(* IEC 61131-3 sources: PortalRobot/Portal_robot/Device/application/FB (part 3) *)

(* ---- FB_ROBOT.st ---- *)
FUNCTION_BLOCK FB_ROBOT
VAR_INPUT

	stMachine_1_Command : ST_ROBOT_COMMAND; // Команда роботу от первого станка
	stMachine_2_Command : ST_ROBOT_COMMAND; // Команда роботу от второго станка
	stMachine_3_Command : ST_ROBOT_COMMAND; // Команда роботу от третьего станка
	stMagazineCommand   : ST_ROBOT_COMMAND; // Команда роботу от магазина
	stCellCommand       : ST_ROBOT_COMMAND; // Команда позиционирования от менеджера ячейки
	stHmiCommand        : ST_ROBOT_COMMAND; // Ручная команда роботу с HMI
	xReset              : BOOL; // Сброс ошибок робота
    xMode               : BOOL; // Режим робота: TRUE — Modbus, FALSE — SoftMotion
	xManual      		: BOOL; // 1 - ручной режим работы, 0 - автоматический режим работы
	xGlobalError        : BOOL; // Глобальная ошибка ячейки
	xModbusBusy         : BOOL; // Внешний робот выполняет команду
	xModbusDone         : BOOL; // Внешний робот завершил команду
	xModbusError        : BOOL; // Ошибка обмена или внешнего робота

    stPoint : ARRAY [0..GVL_POINT.iPointNumber] OF ST_POINT; // Глобальная таблица точек робота

    xSimBlankAvailable : BOOL; // Начальное наличие заготовки в модели захвата

END_VAR
VAR_OUTPUT
	Command       : ST_ROBOT_COMMAND; // Выбранная команда текущего цикла
	ModbusCommand : ST_ROBOT_COMMAND; // Команда внешнему роботу по Modbus
	Status        : ST_ROBOT_STATUS; // Рабочие статусы робота
	Diag          : ST_ROBOT_DIAG; // Состояние автомата и активная команда
	Error         : ST_ROBOT_ERRORS; // Активные и последние ошибки
	GripperDiag   : ST_GRIPPER_DIAG; // Диагностика внутреннего блока захвата
	GripperError  : ST_GRIPPER_ERRORS; // Активные и последние ошибки захвата
END_VAR
VAR
	fbMotionManager  : FB_MOTION_MANAGER; // Менеджер перемещения по точкам
    fbGripper        : FB_GRIPPER_SIMULATION; // Модель двухпозиционного захвата
	stGripperCommand : ST_GRIPPER_COMMAND; // Команда внутренней модели захвата

    eState        : E_ROBOT_STATE := E_ROBOT_STATE.IDLE; // Текущее состояние автомата робота
    eActiveAction : E_ROBOT_ACTION := E_ROBOT_ACTION.NONE; // Защёлкнутое действие
    eActivePoint  : E_POINT_NAME; // Защёлкнутая целевая точка

    xMotionExecute  : BOOL; // Запрос выполнения перемещения
    xGripperExecute : BOOL; // Запрос выполнения действия захвата
	xMagazineCommandActive : BOOL; // Активная команда получена от FB_MAGAZINE

END_VAR

VAR_IN_OUT
    stMotionManager : ST_MOTION_MANAGER; // Данные менеджера движения
    GroupData       : ST_AXIS_GROUP; // Данные группы осей XYZ
    stPointManager  : ST_POINT_MANAGER; // Данные проверки точки
END_VAR

VAR CONSTANT
	ERR_ROBOT_WRONG_ACTION : DWORD := DWORD#16#0000_0001; // Недопустимое действие робота
    ERR_ROBOT_MOTION       : DWORD := DWORD#16#0000_0002; // Ошибка менеджера движения
    ERR_ROBOT_GRIPPER      : DWORD := DWORD#16#0000_0004; // Ошибка захвата
    ERR_ROBOT_MODBUS_STUB  : DWORD := DWORD#16#0000_0008; // Ошибка внешнего робота или Modbus
    ERR_ROBOT_STOP         : DWORD := DWORD#16#0000_0010; // Остановка команды робота
	MASK_LOCAL_ERROR         : DWORD := ERR_ROBOT_WRONG_ACTION OR ERR_ROBOT_MODBUS_STUB; // Собственные первопричины робота
END_VAR

// --- BEGIN IMPLEMENTATION ---

// Команды по умолчанию
xMotionExecute := FALSE;
xGripperExecute := FALSE;
xMagazineCommandActive := FALSE;

Command.xExecute := FALSE;
Command.xStop := FALSE;
Command.xReset := FALSE;
Command.eAction := E_ROBOT_ACTION.NONE;
Command.eSetPoint := E_POINT_NAME.NONE;
Command.iTakeSlot := 0;
Command.iPutSlot := 0;

ModbusCommand.xExecute := FALSE;
ModbusCommand.xStop := FALSE;
ModbusCommand.xReset := xReset;
ModbusCommand.eAction := E_ROBOT_ACTION.NONE;
ModbusCommand.eSetPoint := E_POINT_NAME.NONE;
ModbusCommand.iTakeSlot := 0;
ModbusCommand.iPutSlot := 0;

//Определяем какой режим работы активен
IF NOT xManual THEN
	IF stCellCommand.xExecute OR stCellCommand.xStop THEN
		Command := stCellCommand;
	ELSIF stMachine_1_Command.xExecute THEN
		Command := stMachine_1_Command;
	ELSIF stMachine_2_Command.xExecute THEN
		Command := stMachine_2_Command;
	ELSIF stMachine_3_Command.xExecute THEN
		Command := stMachine_3_Command;
	ELSIF stMagazineCommand.xExecute OR stMagazineCommand.xStop THEN
		Command := stMagazineCommand;
		xMagazineCommandActive := TRUE;
	END_IF
ELSE
	IF stMagazineCommand.xExecute OR stMagazineCommand.xStop THEN
		Command := stMagazineCommand;
		xMagazineCommandActive := TRUE;
	ELSE
		Command := stHmiCommand;
	END_IF
END_IF;

Command.xReset := xReset;

// =====================================================
// Автомат FB_ROBOT
// =====================================================

CASE eState OF

    E_ROBOT_STATE.IDLE:

        Status.xBusy := FALSE;
        Status.xDone := FALSE;
        Status.xError := FALSE;

        IF Command.xExecute
		AND (xMagazineCommandActive
			OR ((Command.eSetPoint <> E_POINT_NAME.MAGAZINE_TAKE_DETAIL)
				AND (Command.eSetPoint <> E_POINT_NAME.MAGAZINE_PUT_DETAIL)
				AND (Command.eSetPoint <> E_POINT_NAME.MAGAZINE_CHANGE_DETAIL))) THEN
            eActiveAction := Command.eAction;
            eActivePoint := Command.eSetPoint;

            IF xMode THEN
                eState := E_ROBOT_STATE.MODBUS_STUB;

            ELSE
                CASE Command.eAction OF

                    E_ROBOT_ACTION.MOVE_TO_POINT:
                        eState := E_ROBOT_STATE.MOTION;

                    E_ROBOT_ACTION.UNCLAMP_1,
                    E_ROBOT_ACTION.CLAMP_1,
                    E_ROBOT_ACTION.UNCLAMP_2,
                    E_ROBOT_ACTION.CLAMP_2,
                    E_ROBOT_ACTION.ROTATE_TO_BLANK,
                    E_ROBOT_ACTION.ROTATE_TO_DETAIL:
                        eState := E_ROBOT_STATE.GRIPPER;

                ELSE
                    Error.dwErrorActive :=
                        Error.dwErrorActive OR ERR_ROBOT_WRONG_ACTION;

                    eState := E_ROBOT_STATE.ERROR;
                END_CASE;
            END_IF;
        END_IF;

    E_ROBOT_STATE.MOTION:

        Status.xBusy := TRUE;
        xMotionExecute := TRUE;

        IF Command.xStop OR xGlobalError THEN
            Error.dwErrorActive := Error.dwErrorActive OR ERR_ROBOT_STOP;
            eState := E_ROBOT_STATE.ERROR;

        ELSIF stMotionManager.Status.xError THEN
            Error.dwErrorActive := Error.dwErrorActive OR ERR_ROBOT_MOTION;
            eState := E_ROBOT_STATE.ERROR;

        ELSIF stMotionManager.Status.xDone THEN
            eState := E_ROBOT_STATE.DONE;
        END_IF;

    E_ROBOT_STATE.GRIPPER:

        Status.xBusy := TRUE;
        xGripperExecute := TRUE;

        IF Command.xStop OR xGlobalError THEN
            Error.dwErrorActive := Error.dwErrorActive OR ERR_ROBOT_STOP;
            eState := E_ROBOT_STATE.ERROR;

        ELSIF fbGripper.Status.xError THEN
            Error.dwErrorActive := Error.dwErrorActive OR ERR_ROBOT_GRIPPER;
            eState := E_ROBOT_STATE.ERROR;

        ELSIF fbGripper.Status.xDone THEN
            eState := E_ROBOT_STATE.DONE;
        END_IF;

    E_ROBOT_STATE.DONE:

        Status.xBusy := FALSE;
        Status.xDone := TRUE;

        CASE eActiveAction OF

            E_ROBOT_ACTION.MOVE_TO_POINT:
                xMotionExecute := TRUE;

            E_ROBOT_ACTION.UNCLAMP_1,
            E_ROBOT_ACTION.CLAMP_1,
            E_ROBOT_ACTION.UNCLAMP_2,
            E_ROBOT_ACTION.CLAMP_2,
            E_ROBOT_ACTION.ROTATE_TO_BLANK,
            E_ROBOT_ACTION.ROTATE_TO_DETAIL:
                xGripperExecute := TRUE;

        END_CASE;

        IF NOT Command.xExecute THEN
            Status.xDone := FALSE;
            eActiveAction := E_ROBOT_ACTION.NONE;
            eState := E_ROBOT_STATE.IDLE;
        END_IF;

    E_ROBOT_STATE.MODBUS_STUB:
		Status.xBusy := TRUE;
		ModbusCommand := Command;
		ModbusCommand.xExecute := TRUE;

		IF Command.xStop OR xGlobalError THEN
			ModbusCommand.xStop := TRUE;
			Error.dwErrorActive := Error.dwErrorActive OR ERR_ROBOT_STOP;
			eState := E_ROBOT_STATE.ERROR;
		ELSIF xModbusError THEN
			Error.dwErrorActive := Error.dwErrorActive OR ERR_ROBOT_MODBUS_STUB;
			eState := E_ROBOT_STATE.ERROR;
		ELSIF xModbusDone THEN
			eState := E_ROBOT_STATE.DONE;
		END_IF;

    E_ROBOT_STATE.ERROR:

        Status.xBusy := FALSE;
        Status.xDone := FALSE;
        Status.xError := TRUE;

        IF xReset
        AND NOT Command.xExecute
        AND NOT Command.xStop
        AND NOT xGlobalError
        AND NOT stMotionManager.Status.xError
		AND NOT fbGripper.Status.xError
		AND NOT xModbusError THEN

			Error.dwErrorLast := Error.dwErrorActive;
            Error.dwErrorActive := DWORD#0;
            Status.xError := FALSE;
            eActiveAction := E_ROBOT_ACTION.NONE;
            eState := E_ROBOT_STATE.IDLE;
        END_IF;

END_CASE;

// =====================================================
// Формирование команды FB_MOTION_MANAGER
// =====================================================

stMotionManager.Command.xExecute := xMotionExecute;
stMotionManager.Command.eTargetPoint := eActivePoint;
stMotionManager.Command.xReset := xReset;

// В ST_MOTION_MANAGER_COMMAND нет отдельного xStop.
// Поэтому Stop передаётся как ошибка верхнего уровня.
stMotionManager.Command.xGlobalError :=
    xGlobalError OR Command.xStop;

// =====================================================
// Вызов FB_MOTION_MANAGER
// =====================================================

fbMotionManager(
    stPoint := stPoint,
    xReset := xReset,
    stMotionManager := stMotionManager,
    GroupData := GroupData,
    stPointManager := stPointManager
);

// =====================================================
// Вызов FB_GRIPPER
// =====================================================

stGripperCommand.xExecute := xGripperExecute;
stGripperCommand.xReset := xReset;
stGripperCommand.eAction := eActiveAction;

fbGripper(
	Command := stGripperCommand,
	Diag => GripperDiag,
	Error => GripperError
);

// =====================================================
// Общие статусы
// =====================================================

Status.eCurrentPoint := stMotionManager.Status.eCurrentPoint;
Status.xGripper1Open :=
    fbGripper.Status.xGripper1Open;

Status.xGripper1Closed :=
    fbGripper.Status.xGripper1Closed;

Status.xGripper2Open :=
    fbGripper.Status.xGripper2Open;

Status.xGripper2Closed :=
    fbGripper.Status.xGripper2Closed;

Status.xRotatedToBlank :=
    fbGripper.Status.xRotatedToBlank;

Status.xRotatedToDetail :=
    fbGripper.Status.xRotatedToDetail;

Status.xBlankAvailable := Status.xGripper1Closed;
Status.xDetailAvailable := Status.xGripper2Closed;

Diag.eState := eState;
Diag.eActiveAction := eActiveAction;
Diag.eActivePoint := eActivePoint;
Error.dwAlarmActive := Error.dwErrorActive AND MASK_LOCAL_ERROR;
Status.xExternalError := (Error.dwErrorActive AND (ERR_ROBOT_MOTION OR ERR_ROBOT_GRIPPER)) <> DWORD#0;

IF Error.dwErrorActive <> DWORD#0 THEN
	Error.dwErrorLast := Error.dwErrorActive;
END_IF;

Error.stErrorActive := UpdateErrorView(dwError := Error.dwErrorActive);
Error.stErrorLast := UpdateErrorView(dwError := Error.dwErrorLast);

(* ---- FB_ROBOT_MODBUS.st ---- *)
{attribute 'no_assign'}
FUNCTION_BLOCK FB_ROBOT_MODBUS
VAR_INPUT
	xEnable          : BOOL; // Применён режим MODBUS_TCP
	xReconnect       : BOOL; // Настройки изменены, выполнить reconnect
	Config           : ST_ROBOT_MODBUS_CONFIG;
	Command          : ST_ROBOT_COMMAND; // Семантическая команда FB_ROBOT
END_VAR
VAR_OUTPUT
	Status           : ST_ROBOT_MODBUS_STATUS;
END_VAR
VAR_IN_OUT
	auiWriteRegisters : ARRAY [0..8] OF UINT; // Документные адреса 1001..1009
	auiReadRegisters  : ARRAY [0..16] OF UINT; // Документные адреса 1101..1117
END_VAR
VAR
	{attribute 'no_assign'}
	fbClient       : ModbusFB.ClientTCP;
	fbRead         : ModbusFB.ClientRequestReadHoldingRegisters;
	fbWrite        : ModbusFB.ClientRequestWriteMultipleRegisters;
	eState         : E_ROBOT_MODBUS_CLIENT_STATE := E_ROBOT_MODBUS_CLIENT_STATE.DISABLED;
	xConnect       : BOOL;
	xReadExecute   : BOOL;
	xWriteExecute  : BOOL;
	xStatusFresh   : BOOL;
	xCommandArmed  : BOOL;
	xCommandActive : BOOL;
	xWritePending  : BOOL;
	xHeartbeatChanged : BOOL;
	xHeartbeatSeen : BOOL;
	xPlcHeartbeatDue : BOOL;
	xStopPending   : BOOL;
	xResetPending  : BOOL;
	xControlClearPending : BOOL;
	rtStop         : R_TRIG;
	rtReset        : R_TRIG;
	rtReconnect    : R_TRIG;
	tonPoll        : TON;
	tonPlcHeartbeat: TON;
	tonRobotHeartbeat : TON;
	tonCommunicationGrace : TON;
	tonCommandTimeout : TON;
	tonReconnect   : TON;
	uiCommandSeq   : UINT;
	uiActiveSeq    : UINT;
	uiDecodedRobotHeartbeat : UINT; // Heartbeat из последнего завершённого FC03
	uiPositionXHigh : UINT; // Координаты из того же завершённого FC03-снимка
	uiPositionXLow  : UINT;
	uiPositionYHigh : UINT;
	uiPositionYLow  : UINT;
	uiPositionZHigh : UINT;
	uiPositionZLow  : UINT;
	uiPlcHeartbeat : UINT;
	uiLastRobotHeartbeat : UINT;
	uiCommandCode  : UINT;
	uiRegisterIndex : UINT;
	dwPositionRaw  : DWORD;
	diPositionRaw  : DINT;
	udiReplyTimeoutUs : UDINT;
END_VAR
VAR CONSTANT
	COMMAND_START_ITEM : UINT := UINT#1000; // Документный 1001
	STATUS_START_ITEM  : UINT := UINT#1100; // Документный 1101
	COMMAND_QUANTITY   : UINT := UINT#9;
	STATUS_QUANTITY    : UINT := UINT#17;
	PROTOCOL_VERSION   : UINT := UINT#3;
	STATUS_CONTROLLER_ON  : UINT := UINT#16#0001;
	STATUS_AUTOMATIC_MODE : UINT := UINT#16#0002;
	STATUS_REMOTE_ENABLED : UINT := UINT#16#0004;
	STATUS_DRIVES_ENABLED : UINT := UINT#16#0008;
	STATUS_HOMED          : UINT := UINT#16#0010;
	STATUS_EMERGENCY_STOP : UINT := UINT#16#0020;
	STATUS_ROBOT_ALARM    : UINT := UINT#16#0040;
	STATUS_ROBOT_READY    : UINT := UINT#16#0080;
	STATUS_POSITION_VALID : UINT := UINT#16#0100;
	STATUS_SIMULATOR_ACTIVE : UINT := UINT#16#0200;
END_VAR

// --- BEGIN IMPLEMENTATION ---

Status.xConfigValid := (Config.aIpAddress[0] > BYTE#0)
	AND (Config.aIpAddress[0] < BYTE#224)
	AND (Config.uiPort > UINT#0)
	AND (Config.uiUnitId <= UINT#255)
	AND (Config.tResponseTimeout >= T#50MS)
	AND (Config.tPollInterval >= T#10MS)
	AND (Config.tHeartbeatTimeout >= T#500MS)
	AND (Config.tCommandTimeout >= T#1S);

	udiReplyTimeoutUs := TIME_TO_UDINT(Config.tResponseTimeout) * UDINT#1000;
	rtStop(CLK := Command.xStop);
	rtReset(CLK := Command.xReset);
	rtReconnect(CLK := xReconnect);
	IF rtStop.Q THEN
		xStopPending := TRUE;
	END_IF;
	IF rtReset.Q THEN
		xResetPending := TRUE;
	END_IF;
xReadExecute := FALSE;
xWriteExecute := FALSE;
xHeartbeatChanged := FALSE;

fbClient(
	xConnect := xConnect,
	aIPaddr := Config.aIpAddress,
	uiPort := Config.uiPort,
	tConnnectTimeOut := Config.tHeartbeatTimeout
);

IF NOT xEnable OR NOT Status.xConfigValid THEN
	xConnect := FALSE;
	eState := E_ROBOT_MODBUS_CLIENT_STATE.DISABLED;
	xStatusFresh := FALSE;
	xCommandArmed := FALSE;
	xCommandActive := FALSE;
	xWritePending := FALSE;
	xStopPending := FALSE;
	xResetPending := FALSE;
	xControlClearPending := FALSE;
	xHeartbeatSeen := FALSE;
	xPlcHeartbeatDue := FALSE;
	uiActiveSeq := UINT#0;
	Status.xConnected := FALSE;
ELSE
	xConnect := TRUE;
	IF rtReconnect.Q THEN
		xConnect := FALSE;
		eState := E_ROBOT_MODBUS_CLIENT_STATE.RECONNECT_WAIT;
		xStatusFresh := FALSE;
		xCommandArmed := FALSE;
		xCommandActive := FALSE;
		xWritePending := FALSE;
		xControlClearPending := FALSE;
		xHeartbeatSeen := FALSE;
		xPlcHeartbeatDue := FALSE;
	END_IF;
END_IF;

CASE eState OF
	E_ROBOT_MODBUS_CLIENT_STATE.DISABLED:
		IF xEnable AND Status.xConfigValid THEN
			xConnect := TRUE;
			eState := E_ROBOT_MODBUS_CLIENT_STATE.CONNECTING;
		END_IF;

	E_ROBOT_MODBUS_CLIENT_STATE.CONNECTING:
		IF fbClient.xConnected THEN
			eState := E_ROBOT_MODBUS_CLIENT_STATE.INITIAL_READ;
		ELSIF fbClient.xError THEN
			Status.udiClientError := TO_UDINT(fbClient.eErrorID);
			xConnect := FALSE;
			eState := E_ROBOT_MODBUS_CLIENT_STATE.RECONNECT_WAIT;
		END_IF;

	E_ROBOT_MODBUS_CLIENT_STATE.INITIAL_READ:
		xReadExecute := TRUE;
		IF fbRead.xDone THEN
			xStatusFresh := TRUE;
			uiCommandSeq := auiReadRegisters[0];
			uiActiveSeq := UINT#0;
			uiPlcHeartbeat := UINT#0;
			uiLastRobotHeartbeat := auiReadRegisters[6];
			xHeartbeatSeen := FALSE;
			FOR uiRegisterIndex := UINT#0 TO UINT#8 DO
				auiWriteRegisters[uiRegisterIndex] := UINT#0;
			END_FOR;
			auiWriteRegisters[7] := uiCommandSeq;
			eState := E_ROBOT_MODBUS_CLIENT_STATE.INITIAL_READ_RELEASE;
		ELSIF fbRead.xError THEN
			Status.udiReadError := TO_UDINT(fbRead.eErrorID);
			xConnect := FALSE;
			eState := E_ROBOT_MODBUS_CLIENT_STATE.RECONNECT_WAIT;
		END_IF;

	E_ROBOT_MODBUS_CLIENT_STATE.INITIAL_READ_RELEASE:
		IF NOT fbRead.xBusy THEN
			eState := E_ROBOT_MODBUS_CLIENT_STATE.CLEAR_COMMAND;
		END_IF;

	E_ROBOT_MODBUS_CLIENT_STATE.CLEAR_COMMAND:
		xWriteExecute := TRUE;
		IF fbWrite.xDone THEN
			eState := E_ROBOT_MODBUS_CLIENT_STATE.CLEAR_COMMAND_RELEASE;
		ELSIF fbWrite.xError THEN
			Status.udiWriteError := TO_UDINT(fbWrite.eErrorID);
			xConnect := FALSE;
			eState := E_ROBOT_MODBUS_CLIENT_STATE.RECONNECT_WAIT;
		END_IF;

	E_ROBOT_MODBUS_CLIENT_STATE.CLEAR_COMMAND_RELEASE:
		IF NOT fbWrite.xBusy THEN
			xCommandArmed := NOT Command.xExecute;
			xCommandActive := FALSE;
			eState := E_ROBOT_MODBUS_CLIENT_STATE.READY;
		END_IF;

	E_ROBOT_MODBUS_CLIENT_STATE.READY:
		IF NOT fbClient.xConnected OR fbClient.xError THEN
			Status.udiClientError := TO_UDINT(fbClient.eErrorID);
			xConnect := FALSE;
			eState := E_ROBOT_MODBUS_CLIENT_STATE.RECONNECT_WAIT;
		ELSIF xStopPending THEN
			// Stop always preempts Reset and normal commands.
			// Execute снимается сразу: после принятого CommandSeq это не отменяет
			// команду, зато позволяет роботу выйти из DONE/ERROR/STOPPED в IDLE.
			// Без этого уже завершённая дискретная команда навечно удерживала
			// Execute=1, а xControlClearPending ждал недостижимый IDLE.
			auiWriteRegisters[0] := UINT#0;
			auiWriteRegisters[1] := UINT#0;
			auiWriteRegisters[2] := UINT#1;
			auiWriteRegisters[3] := UINT#0;
			auiWriteRegisters[4] := UINT#0;
			auiWriteRegisters[5] := UINT#0;
			auiWriteRegisters[6] := UINT#0;
			xStopPending := FALSE;
			xResetPending := FALSE;
			xControlClearPending := TRUE;
			xWritePending := TRUE;
		ELSIF xResetPending THEN
			// Reset обязан прервать незавершённую очистку Stop. Иначе
			// xControlClearPending имеет приоритет и защёлкнутый Reset никогда
			// не попадает в регистр 1004.
			auiWriteRegisters[0] := UINT#0;
			auiWriteRegisters[1] := UINT#0;
			auiWriteRegisters[2] := UINT#0;
			auiWriteRegisters[3] := UINT#1;
			auiWriteRegisters[4] := UINT#0;
			auiWriteRegisters[5] := UINT#0;
			auiWriteRegisters[6] := UINT#0;
			xCommandActive := FALSE;
			uiActiveSeq := UINT#0;
			xCommandArmed := FALSE;
			xResetPending := FALSE;
			xControlClearPending := TRUE;
			xWritePending := TRUE;
		ELSIF xControlClearPending THEN
			// Stop удерживается до STOPPED/IDLE, Reset — до снятия аварии. Так
			// импульс не потеряется между более медленными циклами программы робота.
			IF ((auiWriteRegisters[2] = UINT#1)
				AND ((Status.uiExecutionState = TO_UINT(E_ROBOT_MODBUS_EXECUTION_STATE.STOPPED))
					OR (Status.uiExecutionState = TO_UINT(E_ROBOT_MODBUS_EXECUTION_STATE.IDLE))))
			OR ((auiWriteRegisters[3] = UINT#1)
				AND NOT Status.xRobotAlarm
				AND (Status.uiExecutionState =
					TO_UINT(E_ROBOT_MODBUS_EXECUTION_STATE.IDLE))) THEN
				auiWriteRegisters[2] := UINT#0;
				auiWriteRegisters[3] := UINT#0;
				xCommandActive := FALSE;
				uiActiveSeq := UINT#0;
				// Верхний FB удерживает Execute до появления Busy. Поэтому после
				// подтверждённой очистки принимаем уже удерживаемую новую команду,
				// а не требуем ещё одного фронта от HMI.
				xCommandArmed := TRUE;
				xControlClearPending := FALSE;
				xWritePending := TRUE;
			END_IF;
		ELSIF Command.xExecute AND xCommandArmed AND NOT xCommandActive THEN
			uiCommandCode := UINT#0;
			CASE Command.eAction OF
				E_ROBOT_ACTION.MOVE_TO_POINT:
					CASE Command.eSetPoint OF
						E_POINT_NAME.MACHINE_1_ABOVE: uiCommandCode := UINT#10;
						E_POINT_NAME.MACHINE_1_INSIDE: uiCommandCode := UINT#11;
						E_POINT_NAME.MACHINE_1_CHUCK_APROACH: uiCommandCode := UINT#12;
						E_POINT_NAME.MACHINE_1_CHUCK_POSITION: uiCommandCode := UINT#13;
						E_POINT_NAME.MACHINE_2_ABOVE: uiCommandCode := UINT#14;
						E_POINT_NAME.MACHINE_2_INSIDE: uiCommandCode := UINT#15;
						E_POINT_NAME.MACHINE_2_CHUCK_APROACH: uiCommandCode := UINT#16;
						E_POINT_NAME.MACHINE_2_CHUCK_POSITION: uiCommandCode := UINT#17;
						E_POINT_NAME.MACHINE_3_ABOVE: uiCommandCode := UINT#18;
						E_POINT_NAME.MACHINE_3_INSIDE: uiCommandCode := UINT#19;
						E_POINT_NAME.MACHINE_3_CHUCK_APROACH: uiCommandCode := UINT#20;
						E_POINT_NAME.MACHINE_3_CHUCK_POSITION: uiCommandCode := UINT#21;
						E_POINT_NAME.HOME_SAFETY: uiCommandCode := UINT#22;
						E_POINT_NAME.MAGAZINE_SAFE: uiCommandCode := UINT#23;
						E_POINT_NAME.MAGAZINE_CHANGE: uiCommandCode := UINT#24;
						E_POINT_NAME.MAGAZINE_IN_SLOT: uiCommandCode := UINT#25;
					END_CASE;
				E_ROBOT_ACTION.UNCLAMP_1: uiCommandCode := UINT#2;
				E_ROBOT_ACTION.CLAMP_1: uiCommandCode := UINT#3;
				E_ROBOT_ACTION.UNCLAMP_2: uiCommandCode := UINT#4;
				E_ROBOT_ACTION.CLAMP_2: uiCommandCode := UINT#5;
				E_ROBOT_ACTION.ROTATE_TO_BLANK: uiCommandCode := UINT#6;
				E_ROBOT_ACTION.ROTATE_TO_DETAIL: uiCommandCode := UINT#7;
			END_CASE;

			IF uiCommandCode > UINT#0 THEN
				uiCommandSeq := uiCommandSeq + UINT#1;
				IF uiCommandSeq = UINT#0 THEN
					uiCommandSeq := UINT#1;
				END_IF;
				uiActiveSeq := uiCommandSeq;
				auiWriteRegisters[0] := uiCommandCode;
				auiWriteRegisters[1] := UINT#1;
				auiWriteRegisters[2] := UINT#0;
				auiWriteRegisters[3] := UINT#0;
				auiWriteRegisters[4] := SINT_TO_UINT(Command.iActiveSlot);
				auiWriteRegisters[5] := Command.uiMagazineId;
				auiWriteRegisters[6] := UINT#0;
				auiWriteRegisters[7] := uiCommandSeq;
				xCommandActive := TRUE;
				xCommandArmed := FALSE;
				xWritePending := TRUE;
			END_IF;
		ELSIF NOT Command.xExecute AND xCommandActive THEN
			auiWriteRegisters[0] := UINT#0;
			auiWriteRegisters[1] := UINT#0;
			auiWriteRegisters[2] := UINT#0;
			auiWriteRegisters[3] := UINT#0;
			auiWriteRegisters[4] := UINT#0;
			auiWriteRegisters[5] := UINT#0;
			auiWriteRegisters[6] := UINT#0;
			xCommandActive := FALSE;
			// CommandSeq в регистре сохраняется как последний использованный номер,
			// но завершённая транзакция больше не имеет права публиковать Done.
			// Повтор после Reset всегда получит новый ненулевой sequence.
			uiActiveSeq := UINT#0;
			xCommandArmed := TRUE;
			xWritePending := TRUE;
		ELSIF NOT Command.xExecute THEN
			xCommandArmed := TRUE;
		END_IF;

		IF xPlcHeartbeatDue THEN
			uiPlcHeartbeat := uiPlcHeartbeat + UINT#1;
			auiWriteRegisters[8] := uiPlcHeartbeat;
			xPlcHeartbeatDue := FALSE;
			xWritePending := TRUE;
		END_IF;

		IF xWritePending THEN
			eState := E_ROBOT_MODBUS_CLIENT_STATE.WRITE_COMMAND;
		ELSIF tonPoll.Q THEN
			eState := E_ROBOT_MODBUS_CLIENT_STATE.READ_STATUS;
		END_IF;

	E_ROBOT_MODBUS_CLIENT_STATE.WRITE_COMMAND:
		xWriteExecute := TRUE;
		IF fbWrite.xDone THEN
			xWritePending := FALSE;
			eState := E_ROBOT_MODBUS_CLIENT_STATE.WRITE_COMMAND_RELEASE;
		ELSIF fbWrite.xError THEN
			Status.udiWriteError := TO_UDINT(fbWrite.eErrorID);
			xConnect := FALSE;
			eState := E_ROBOT_MODBUS_CLIENT_STATE.RECONNECT_WAIT;
		END_IF;

	E_ROBOT_MODBUS_CLIENT_STATE.WRITE_COMMAND_RELEASE:
		IF NOT fbWrite.xBusy THEN
			eState := E_ROBOT_MODBUS_CLIENT_STATE.READ_STATUS;
		END_IF;

	E_ROBOT_MODBUS_CLIENT_STATE.READ_STATUS:
		xReadExecute := TRUE;
		IF fbRead.xDone THEN
			xStatusFresh := TRUE;
			eState := E_ROBOT_MODBUS_CLIENT_STATE.READ_STATUS_RELEASE;
		ELSIF fbRead.xError THEN
			Status.udiReadError := TO_UDINT(fbRead.eErrorID);
			xConnect := FALSE;
			eState := E_ROBOT_MODBUS_CLIENT_STATE.RECONNECT_WAIT;
		END_IF;

	E_ROBOT_MODBUS_CLIENT_STATE.READ_STATUS_RELEASE:
		IF NOT fbRead.xBusy THEN
			eState := E_ROBOT_MODBUS_CLIENT_STATE.READY;
		END_IF;

	E_ROBOT_MODBUS_CLIENT_STATE.RECONNECT_WAIT:
		xConnect := FALSE;
		xStatusFresh := FALSE;
		IF tonReconnect.Q THEN
			xConnect := TRUE;
			eState := E_ROBOT_MODBUS_CLIENT_STATE.CONNECTING;
		END_IF;
END_CASE;

fbRead(
	xExecute := xReadExecute,
	udiTimeOut := udiReplyTimeoutUs,
	rClient := fbClient,
	uiUnitId := Config.uiUnitId,
	udiReplyTimeout := udiReplyTimeoutUs,
	uiMaxRetries := UINT#1,
	uiStartItem := STATUS_START_ITEM,
	uiQuantity := STATUS_QUANTITY,
	pData := ADR(auiReadRegisters)
);
fbWrite(
	xExecute := xWriteExecute,
	udiTimeOut := udiReplyTimeoutUs,
	rClient := fbClient,
	uiUnitId := Config.uiUnitId,
	udiReplyTimeout := udiReplyTimeoutUs,
	uiMaxRetries := UINT#1,
	uiStartItem := COMMAND_START_ITEM,
	uiQuantity := COMMAND_QUANTITY,
	pData := ADR(auiWriteRegisters)
);

// FC03 может завершиться внутри вызова fbRead. Декодирование выполняется после
// вызова, чтобы технологический Status и сырые диагностические регистры всегда
// относились к одному и тому же снимку опроса.
IF fbRead.xDone THEN
	Status.uiAckSeq := auiReadRegisters[0];
	Status.uiExecutionState := auiReadRegisters[1];
	Status.uiResultCode := auiReadRegisters[2];
	Status.uiActiveCommand := auiReadRegisters[3];
	Status.uiCurrentPoint := auiReadRegisters[4];
	Status.uiGripperStatus := auiReadRegisters[5];
	Status.uiRobotHeartbeat := auiReadRegisters[6];
	Status.uiStatusWord := auiReadRegisters[7];
	Status.uiAlarmCode := auiReadRegisters[8];
	Status.uiOperationPhase := auiReadRegisters[15];
	Status.uiProtocolVersion := auiReadRegisters[16];
	uiDecodedRobotHeartbeat := auiReadRegisters[6];
	uiPositionXHigh := auiReadRegisters[9];
	uiPositionXLow := auiReadRegisters[10];
	uiPositionYHigh := auiReadRegisters[11];
	uiPositionYLow := auiReadRegisters[12];
	uiPositionZHigh := auiReadRegisters[13];
	uiPositionZLow := auiReadRegisters[14];
END_IF;

tonPoll(IN := eState = E_ROBOT_MODBUS_CLIENT_STATE.READY, PT := Config.tPollInterval);
// Heartbeat timer is independent of request states. The due latch prevents a pulse
// from being lost while FC03/FC16 is busy.
tonPlcHeartbeat(
	IN := xEnable AND fbClient.xConnected AND NOT tonPlcHeartbeat.Q,
	PT := T#100MS
);
IF tonPlcHeartbeat.Q THEN
	xPlcHeartbeatDue := TRUE;
END_IF;
tonReconnect(IN := eState = E_ROBOT_MODBUS_CLIENT_STATE.RECONNECT_WAIT, PT := T#1S);

Status.xConnected := fbClient.xConnected AND xConnect;
Status.xStatusFresh := xStatusFresh;

IF uiDecodedRobotHeartbeat <> uiLastRobotHeartbeat THEN
	uiLastRobotHeartbeat := uiDecodedRobotHeartbeat;
	xHeartbeatChanged := TRUE;
	xHeartbeatSeen := TRUE;
END_IF;
tonRobotHeartbeat(
	IN := xEnable AND xStatusFresh AND NOT xHeartbeatChanged,
	PT := Config.tHeartbeatTimeout
);
Status.xCommunicationAlive := Status.xConnected
	AND xStatusFresh
	AND xHeartbeatSeen
	AND NOT tonRobotHeartbeat.Q
	AND (Status.uiProtocolVersion = PROTOCOL_VERSION);
tonCommunicationGrace(
	IN := xEnable AND Status.xConfigValid AND NOT Status.xCommunicationAlive,
	PT := Config.tHeartbeatTimeout
);

Status.xControllerOn := (Status.uiStatusWord AND STATUS_CONTROLLER_ON) <> UINT#0;
Status.xAutomaticMode := (Status.uiStatusWord AND STATUS_AUTOMATIC_MODE) <> UINT#0;
Status.xRemoteEnabled := (Status.uiStatusWord AND STATUS_REMOTE_ENABLED) <> UINT#0;
Status.xDrivesEnabled := (Status.uiStatusWord AND STATUS_DRIVES_ENABLED) <> UINT#0;
Status.xHomed := (Status.uiStatusWord AND STATUS_HOMED) <> UINT#0;
Status.xEmergencyStop := (Status.uiStatusWord AND STATUS_EMERGENCY_STOP) <> UINT#0;
Status.xRobotAlarm := ((Status.uiStatusWord AND STATUS_ROBOT_ALARM) <> UINT#0)
	OR (Status.uiAlarmCode <> UINT#0);
Status.xPositionValid := (Status.uiStatusWord AND STATUS_POSITION_VALID) <> UINT#0;
Status.xSimulatorActive := (Status.uiStatusWord AND STATUS_SIMULATOR_ACTIVE) <> UINT#0;
Status.xReady := Status.xCommunicationAlive
	AND Status.xControllerOn
	AND Status.xAutomaticMode
	AND Status.xRemoteEnabled
	AND Status.xDrivesEnabled
	AND Status.xHomed
	AND Status.xPositionValid
	AND NOT Status.xEmergencyStop
	AND NOT Status.xRobotAlarm
	AND ((Status.uiStatusWord AND STATUS_ROBOT_READY) <> UINT#0);

Status.xDone := (uiActiveSeq <> UINT#0)
	AND xCommandActive
	AND (Status.uiAckSeq = uiActiveSeq)
	AND (Status.uiExecutionState = TO_UINT(E_ROBOT_MODBUS_EXECUTION_STATE.DONE))
	AND (Status.uiResultCode = UINT#0);
// Busy означает активную PLC-транзакцию, включая ожидание AckSeq. Благодаря
// этому FB_ROBOT обязательно увидит запуск новой команды до её terminal state.
Status.xBusy := (uiActiveSeq <> UINT#0)
	AND xCommandActive
	AND NOT Status.xDone
	AND NOT ((Status.uiAckSeq = uiActiveSeq)
		AND ((Status.uiExecutionState = TO_UINT(E_ROBOT_MODBUS_EXECUTION_STATE.ERROR))
			OR (Status.uiExecutionState = TO_UINT(E_ROBOT_MODBUS_EXECUTION_STATE.STOPPED))
			OR ((Status.uiExecutionState = TO_UINT(E_ROBOT_MODBUS_EXECUTION_STATE.DONE))
				AND (Status.uiResultCode <> UINT#0))));
tonCommandTimeout(
	IN := xCommandActive AND NOT Status.xDone,
	PT := Config.tCommandTimeout
);
Status.xCommandTimeout := tonCommandTimeout.Q;
Status.xError := tonCommunicationGrace.Q
	OR Status.xRobotAlarm
	OR Status.xCommandTimeout
	OR ((uiActiveSeq <> UINT#0)
		AND (Status.uiAckSeq = uiActiveSeq)
		AND ((Status.uiExecutionState = TO_UINT(E_ROBOT_MODBUS_EXECUTION_STATE.ERROR))
			OR ((Status.uiExecutionState = TO_UINT(E_ROBOT_MODBUS_EXECUTION_STATE.DONE))
				AND (Status.uiResultCode <> UINT#0))));

dwPositionRaw := SHL(UINT_TO_DWORD(uiPositionXHigh), 16)
	OR UINT_TO_DWORD(uiPositionXLow);
diPositionRaw := DWORD_TO_DINT(dwPositionRaw);
Status.lrActualX := DINT_TO_LREAL(diPositionRaw) / LREAL#10.0;
dwPositionRaw := SHL(UINT_TO_DWORD(uiPositionYHigh), 16)
	OR UINT_TO_DWORD(uiPositionYLow);
diPositionRaw := DWORD_TO_DINT(dwPositionRaw);
Status.lrActualY := DINT_TO_LREAL(diPositionRaw) / LREAL#10.0;
dwPositionRaw := SHL(UINT_TO_DWORD(uiPositionZHigh), 16)
	OR UINT_TO_DWORD(uiPositionZLow);
diPositionRaw := DWORD_TO_DINT(dwPositionRaw);
Status.lrActualZ := DINT_TO_LREAL(diPositionRaw) / LREAL#10.0;

(* ---- FB_SIMULATION_DYNAMIC_LIMITS.st ---- *)
FUNCTION_BLOCK FB_SIMULATION_DYNAMIC_LIMITS
VAR_INPUT
	xSimulationMode : BOOL; // Активна тестовая среда SIMULATION
	xSoftMotionMode : BOOL; // Роботом управляют локальные оси SoftMotion
	xAccelerationEnabled : BOOL; // Для следующего теста выбран ускоренный профиль
	xPrepareTest : BOOL; // Фронт подготовки следующего сценария
	uiRequestedFactor : UINT; // Запрошенное масштабирование времени 1..100
	xCellRunning : BOOL;
	xRobotBusy : BOOL;
	xMotionBusy : BOOL;
	xDrivesPowered : BOOL;
	xDrivesOff : BOOL;
	eGroupState : E_AXIS_GROUP_STATE;
	tTransactionTimeout : TIME := T#60S; // Общий предел Stop -> Disable -> Change -> Enable
END_VAR
VAR_OUTPUT
	xCellStopRequest : BOOL; // Сначала остановить технологический цикл
	xMotionStopRequest : BOOL; // Затем остановить движение группы
	xGroupDisableRequest : BOOL; // Перед изменением лимитов получить GroupDisabled
	xDrivesEnableRequest : BOOL; // После изменения вернуть штатную готовность
	xBusy : BOOL;
	xPending : BOOL; // Ползунок изменён; значение ждёт границы следующего теста
	xReadyForTest : BOOL; // Новый тест можно запускать
	xAccelerationActive : BOOL;
	uiAppliedFactor : UINT := UINT#1;
	xDone : BOOL;
	xError : BOOL;
	udiErrorId : UDINT;
END_VAR
VAR_IN_OUT
	AxisX : AXIS_REF_SM3;
	AxisY : AXIS_REF_SM3;
	AxisZ : AXIS_REF_SM3;
END_VAR
VAR CONSTANT
	STATE_IDLE : UINT := UINT#0;
	STATE_WAIT_STANDSTILL : UINT := UINT#10;
	STATE_WAIT_GROUP_DISABLED : UINT := UINT#20;
	STATE_CHANGE_X : UINT := UINT#30;
	STATE_CHANGE_Y : UINT := UINT#40;
	STATE_CHANGE_Z : UINT := UINT#50;
	STATE_PREPARE_ROLLBACK : UINT := UINT#55;
	STATE_WAIT_REENABLE : UINT := UINT#60;
	STATE_LOCKED_ERROR : UINT := UINT#90;
	ERR_INVALID_ORIGINAL_LIMITS : UDINT := UDINT#16#80010001;
	ERR_TRANSACTION_TIMEOUT : UDINT := UDINT#16#80010002;
	ERR_INVALID_STATE : UDINT := UDINT#16#80010003;
END_VAR
VAR
	rtPrepareTest : R_TRIG;
	tonTransaction : TON;
	uiState : UINT := UINT#0;
	uiAxis : UINT;
	uiDesiredFactor : UINT := UINT#1;
	uiTargetFactor : UINT := UINT#1;
	xOriginalLimitsSaved : BOOL;
	xOriginalLimitsValid : BOOL;
	xRestoreOnExit : BOOL;
	xRollback : BOOL;
	xReenableAfterChange : BOOL;

	alrOriginalVelocity : ARRAY [1..3] OF LREAL;
	alrOriginalAcceleration : ARRAY [1..3] OF LREAL;
	alrOriginalDeceleration : ARRAY [1..3] OF LREAL;
	alrOriginalJerk : ARRAY [1..3] OF LREAL;
	alrTargetVelocity : ARRAY [1..3] OF LREAL;
	alrTargetAcceleration : ARRAY [1..3] OF LREAL;
	alrTargetDeceleration : ARRAY [1..3] OF LREAL;
	alrTargetJerk : ARRAY [1..3] OF LREAL;
	lrFactor : LREAL;
	lrFactorSquared : LREAL;
	lrFactorCubed : LREAL;

	fbChangeX : SMC_ChangeDynamicLimits;
	fbChangeY : SMC_ChangeDynamicLimits;
	fbChangeZ : SMC_ChangeDynamicLimits;
END_VAR

// --- BEGIN IMPLEMENTATION ---

// Запрошенное значение разрешено менять когда угодно. Оно только создаёт
// pending-запрос; уже выполняемая траектория никогда не перепланируется.
uiDesiredFactor := MAX(UINT#1, MIN(UINT#100, uiRequestedFactor));
IF NOT (xSimulationMode AND xSoftMotionMode AND xAccelerationEnabled) THEN
	uiDesiredFactor := UINT#1;
END_IF;
rtPrepareTest(CLK := xPrepareTest);

xCellStopRequest := FALSE;
xMotionStopRequest := FALSE;
xGroupDisableRequest := FALSE;
xDrivesEnableRequest := FALSE;
xDone := FALSE;

// Штатные лимиты снимаются ровно при входе в SoftMotion-симуляцию, до первого
// масштабирования. Прямое редактирование AXIS_REF здесь не выполняется.
IF xSimulationMode AND xSoftMotionMode AND NOT xOriginalLimitsSaved THEN
	// Dynamic limits из конфигуратора оси находятся в fSWMax*. fMax* — это
	// remote limits самого привода и у виртуальной оси законно остаются нулями.
	alrOriginalVelocity[1] := AxisX.fSWMaxVelocity;
	alrOriginalAcceleration[1] := AxisX.fSWMaxAcceleration;
	alrOriginalDeceleration[1] := AxisX.fSWMaxDeceleration;
	alrOriginalJerk[1] := AxisX.fSWMaxJerk;
	alrOriginalVelocity[2] := AxisY.fSWMaxVelocity;
	alrOriginalAcceleration[2] := AxisY.fSWMaxAcceleration;
	alrOriginalDeceleration[2] := AxisY.fSWMaxDeceleration;
	alrOriginalJerk[2] := AxisY.fSWMaxJerk;
	alrOriginalVelocity[3] := AxisZ.fSWMaxVelocity;
	alrOriginalAcceleration[3] := AxisZ.fSWMaxAcceleration;
	alrOriginalDeceleration[3] := AxisZ.fSWMaxDeceleration;
	alrOriginalJerk[3] := AxisZ.fSWMaxJerk;

	IF alrOriginalVelocity[1] <= LREAL#0.0 THEN alrOriginalVelocity[1] := AxisX.fMaxVelocity; END_IF;
	IF alrOriginalAcceleration[1] <= LREAL#0.0 THEN alrOriginalAcceleration[1] := AxisX.fMaxAcceleration; END_IF;
	IF alrOriginalDeceleration[1] <= LREAL#0.0 THEN alrOriginalDeceleration[1] := AxisX.fMaxDeceleration; END_IF;
	IF alrOriginalJerk[1] <= LREAL#0.0 THEN alrOriginalJerk[1] := AxisX.fMaxJerk; END_IF;
	IF alrOriginalVelocity[2] <= LREAL#0.0 THEN alrOriginalVelocity[2] := AxisY.fMaxVelocity; END_IF;
	IF alrOriginalAcceleration[2] <= LREAL#0.0 THEN alrOriginalAcceleration[2] := AxisY.fMaxAcceleration; END_IF;
	IF alrOriginalDeceleration[2] <= LREAL#0.0 THEN alrOriginalDeceleration[2] := AxisY.fMaxDeceleration; END_IF;
	IF alrOriginalJerk[2] <= LREAL#0.0 THEN alrOriginalJerk[2] := AxisY.fMaxJerk; END_IF;
	IF alrOriginalVelocity[3] <= LREAL#0.0 THEN alrOriginalVelocity[3] := AxisZ.fMaxVelocity; END_IF;
	IF alrOriginalAcceleration[3] <= LREAL#0.0 THEN alrOriginalAcceleration[3] := AxisZ.fMaxAcceleration; END_IF;
	IF alrOriginalDeceleration[3] <= LREAL#0.0 THEN alrOriginalDeceleration[3] := AxisZ.fMaxDeceleration; END_IF;
	IF alrOriginalJerk[3] <= LREAL#0.0 THEN alrOriginalJerk[3] := AxisZ.fMaxJerk; END_IF;

	xOriginalLimitsValid := TRUE;
	FOR uiAxis := UINT#1 TO UINT#3 DO
		xOriginalLimitsValid := xOriginalLimitsValid
			AND (alrOriginalVelocity[uiAxis] > LREAL#0.0)
			AND (alrOriginalAcceleration[uiAxis] > LREAL#0.0)
			AND (alrOriginalDeceleration[uiAxis] > LREAL#0.0)
			AND (alrOriginalJerk[uiAxis] > LREAL#0.0);
	END_FOR;
	IF xOriginalLimitsValid THEN
		xOriginalLimitsSaved := TRUE;
		uiAppliedFactor := UINT#1;
		xError := FALSE;
		udiErrorId := UDINT#0;
	ELSIF rtPrepareTest.Q THEN
		// До подготовки теста просто ждём инициализацию осей; не защёлкиваем
		// ложную ошибку на первом цикле после переключения среды.
		xError := TRUE;
		udiErrorId := ERR_INVALID_ORIGINAL_LIMITS;
	END_IF;
END_IF;

// Ошибка чтения исходных лимитов не должна блокировать обычную ячейку после
// выхода из тестовой среды и не должна переживать Online Change этого исправления.
IF NOT xSimulationMode
AND NOT xOriginalLimitsSaved
AND (uiState = STATE_IDLE)
AND (udiErrorId = ERR_INVALID_ORIGINAL_LIMITS) THEN
	xError := FALSE;
	udiErrorId := UDINT#0;
END_IF;

xRestoreOnExit := xOriginalLimitsSaved
	AND (NOT xSimulationMode OR NOT xSoftMotionMode)
	AND (uiAppliedFactor <> UINT#1);
xPending := xOriginalLimitsSaved AND (uiDesiredFactor <> uiAppliedFactor);

// Один общий таймаут защищает всю транзакцию Stop -> Disable -> Change -> Enable.
tonTransaction(IN := uiState <> STATE_IDLE, PT := tTransactionTimeout);
IF tonTransaction.Q
AND (uiState <> STATE_IDLE)
AND (uiState <> STATE_LOCKED_ERROR) THEN
	xError := TRUE;
	udiErrorId := ERR_TRANSACTION_TIMEOUT;
	uiState := STATE_LOCKED_ERROR;
END_IF;

CASE uiState OF
	STATE_IDLE:
		xBusy := FALSE;
		// Возврат штатных лимитов при выходе из SIMULATION выполняется сразу.
		// Обычная ячейка не получит Start, пока транзакция не закончена.
		IF xRestoreOnExit THEN
			xError := FALSE;
			udiErrorId := UDINT#0;
			uiTargetFactor := UINT#1;
			xRollback := FALSE;
			xReenableAfterChange := xSoftMotionMode AND NOT xDrivesOff;
			xBusy := TRUE;
			uiState := STATE_WAIT_STANDSTILL;
		ELSIF rtPrepareTest.Q
		AND xSimulationMode
		AND xSoftMotionMode
		AND xPending
		AND NOT xCellRunning THEN
			xError := FALSE;
			udiErrorId := UDINT#0;
			uiTargetFactor := uiDesiredFactor;
			xRollback := FALSE;
			xReenableAfterChange := NOT xDrivesOff;
			xBusy := TRUE;
			uiState := STATE_WAIT_STANDSTILL;
		ELSIF NOT xSimulationMode
		AND xOriginalLimitsSaved
		AND (uiAppliedFactor = UINT#1) THEN
			// Лимиты не менялись либо уже успешно восстановлены.
			xOriginalLimitsSaved := FALSE;
		END_IF;

	STATE_WAIT_STANDSTILL:
		xBusy := TRUE;
		xCellStopRequest := xCellRunning;
		xMotionStopRequest := xMotionBusy OR xRobotBusy;
		IF NOT xCellRunning AND NOT xMotionBusy AND NOT xRobotBusy THEN
			uiState := STATE_WAIT_GROUP_DISABLED;
		END_IF;

	STATE_WAIT_GROUP_DISABLED:
		xBusy := TRUE;
		xGroupDisableRequest := NOT xDrivesOff;
		IF xDrivesOff AND (eGroupState = E_AXIS_GROUP_STATE.DISABLED) THEN
			IF xRollback THEN
				FOR uiAxis := UINT#1 TO UINT#3 DO
					alrTargetVelocity[uiAxis] := alrOriginalVelocity[uiAxis];
					alrTargetAcceleration[uiAxis] := alrOriginalAcceleration[uiAxis];
					alrTargetDeceleration[uiAxis] := alrOriginalDeceleration[uiAxis];
					alrTargetJerk[uiAxis] := alrOriginalJerk[uiAxis];
				END_FOR;
			ELSE
				lrFactor := UINT_TO_LREAL(uiTargetFactor);
				lrFactorSquared := lrFactor * lrFactor;
				lrFactorCubed := lrFactorSquared * lrFactor;
				alrTargetVelocity[1] := alrOriginalVelocity[1] * lrFactor;
				alrTargetAcceleration[1] := alrOriginalAcceleration[1] * lrFactorSquared;
				alrTargetDeceleration[1] := alrOriginalDeceleration[1] * lrFactorSquared;
				alrTargetJerk[1] := alrOriginalJerk[1] * lrFactorCubed;
				alrTargetVelocity[2] := alrOriginalVelocity[2] * lrFactor;
				alrTargetAcceleration[2] := alrOriginalAcceleration[2] * lrFactorSquared;
				alrTargetDeceleration[2] := alrOriginalDeceleration[2] * lrFactorSquared;
				alrTargetJerk[2] := alrOriginalJerk[2] * lrFactorCubed;
				alrTargetVelocity[3] := alrOriginalVelocity[3] * lrFactor;
				alrTargetAcceleration[3] := alrOriginalAcceleration[3] * lrFactorSquared;
				alrTargetDeceleration[3] := alrOriginalDeceleration[3] * lrFactorSquared;
				alrTargetJerk[3] := alrOriginalJerk[3] * lrFactorCubed;
			END_IF;
			uiState := STATE_CHANGE_X;
		END_IF;

	STATE_CHANGE_X:
		xBusy := TRUE;
		IF fbChangeX.bError THEN
			xError := TRUE;
			udiErrorId := TO_UDINT(fbChangeX.ErrorID);
			IF xRollback THEN uiState := STATE_LOCKED_ERROR;
			ELSE uiState := STATE_PREPARE_ROLLBACK; END_IF;
		ELSIF fbChangeX.bDone THEN
			uiState := STATE_CHANGE_Y;
		END_IF;

	STATE_CHANGE_Y:
		xBusy := TRUE;
		IF fbChangeY.bError THEN
			xError := TRUE;
			udiErrorId := TO_UDINT(fbChangeY.ErrorID);
			IF xRollback THEN uiState := STATE_LOCKED_ERROR;
			ELSE uiState := STATE_PREPARE_ROLLBACK; END_IF;
		ELSIF fbChangeY.bDone THEN
			uiState := STATE_CHANGE_Z;
		END_IF;

	STATE_CHANGE_Z:
		xBusy := TRUE;
		IF fbChangeZ.bError THEN
			xError := TRUE;
			udiErrorId := TO_UDINT(fbChangeZ.ErrorID);
			IF xRollback THEN uiState := STATE_LOCKED_ERROR;
			ELSE uiState := STATE_PREPARE_ROLLBACK; END_IF;
		ELSIF fbChangeZ.bDone THEN
			IF xReenableAfterChange THEN
				uiState := STATE_WAIT_REENABLE;
			ELSE
				IF xRollback THEN uiAppliedFactor := UINT#1;
				ELSE uiAppliedFactor := uiTargetFactor; END_IF;
				xDone := NOT xRollback;
				xBusy := FALSE;
				uiState := STATE_IDLE;
			END_IF;
		END_IF;

	STATE_PREPARE_ROLLBACK:
		// Один цикл с Execute=FALSE создаёт корректный новый фронт для X.
		xBusy := TRUE;
		xRollback := TRUE;
		uiState := STATE_WAIT_GROUP_DISABLED;

	STATE_WAIT_REENABLE:
		xBusy := TRUE;
		xDrivesEnableRequest := TRUE;
		IF xDrivesPowered AND (eGroupState = E_AXIS_GROUP_STATE.READY) THEN
			IF xRollback THEN uiAppliedFactor := UINT#1;
			ELSE uiAppliedFactor := uiTargetFactor; END_IF;
			xDone := NOT xRollback;
			xBusy := FALSE;
			uiState := STATE_IDLE;
		END_IF;

	STATE_LOCKED_ERROR:
		// При неизвестном/неустранимом результате оставляем группу отключённой.
		// Следующий Start заблокирован, пока инженер не устранит причину.
		xBusy := FALSE;
		xGroupDisableRequest := NOT xDrivesOff;

ELSE
	xError := TRUE;
	udiErrorId := ERR_INVALID_STATE;
	uiState := STATE_LOCKED_ERROR;
END_CASE;

fbChangeX(
	Axis := AxisX,
	bExecute := uiState = STATE_CHANGE_X,
	fMaxVelocity := alrTargetVelocity[1],
	fMaxAcceleration := alrTargetAcceleration[1],
	fMaxDeceleration := alrTargetDeceleration[1],
	fMaxJerk := alrTargetJerk[1]
);
fbChangeY(
	Axis := AxisY,
	bExecute := uiState = STATE_CHANGE_Y,
	fMaxVelocity := alrTargetVelocity[2],
	fMaxAcceleration := alrTargetAcceleration[2],
	fMaxDeceleration := alrTargetDeceleration[2],
	fMaxJerk := alrTargetJerk[2]
);
fbChangeZ(
	Axis := AxisZ,
	bExecute := uiState = STATE_CHANGE_Z,
	fMaxVelocity := alrTargetVelocity[3],
	fMaxAcceleration := alrTargetAcceleration[3],
	fMaxDeceleration := alrTargetDeceleration[3],
	fMaxJerk := alrTargetJerk[3]
);

xPending := xOriginalLimitsSaved AND (uiDesiredFactor <> uiAppliedFactor);
xAccelerationActive := xSimulationMode AND xSoftMotionMode
	AND (uiAppliedFactor > UINT#1) AND NOT xError;
xReadyForTest := NOT xBusy AND NOT xError
	AND (NOT (xSimulationMode AND xSoftMotionMode AND xAccelerationEnabled) OR NOT xPending);

(* ---- FB_TWO_PALLET.st ---- *)
FUNCTION_BLOCK FB_TWO_PALLET
VAR_INPUT
	xSelected : BOOL;
	xManual : BOOL;
	xSafe : BOOL;
	xRobotClear : BOOL; // Окно планировщика и освобождение зоны для обмена в автоматическом режиме
	xRobotIdle : BOOL; // Останов робота без проверки точек, интерфейса и зоны магазина
	xRobotOperation : BOOL; // Текущая или уже выданная операция с этим магазином
	xRobotGeometryReady : BOOL; // Точки робота нужны для работы ячейки, но не для включения магазина
	xRobotMagazineReady : BOOL; // Ошибки и геометрия магазина; содержимое не блокирует включение
	xConnection : BOOL;
	xStopRequest : BOOL;
	xAutoSwap : BOOL;
	xOtherLoaded : BOOL;
	xActivePalletEditAllowed : BOOL;
	xConfigurationChanged : BOOL;
	xExternalCommandRejected : BOOL;
	Command : ST_TWO_PALLET_COMMAND;
	Config : ST_TWO_PALLET_CONFIG;
	Input : ST_TWO_PALLET_INPUT;
END_VAR
VAR_OUTPUT
	Status : ST_TWO_PALLET_STATUS;
	Diag : ST_TWO_PALLET_DIAG;
	Error : ST_TWO_PALLET_ERRORS;
	Output : ST_TWO_PALLET_OUTPUT;
END_VAR
VAR
	ePreviousState : E_TWO_PALLET_STATE := E_TWO_PALLET_STATE.IDLE;
	uiFrom : UINT;
	uiTo : UINT;
	uiSelected : UINT;
	uiCandidate : UINT;
	uiPreviousCandidate : UINT;
	uiConfirmedCandidate : UINT;
	uiManualSelected : UINT;
	uiJogDirection : UINT;
	uiSignals : UINT;
	uiSelectedSignals : UINT;
	uiTargetSignals : UINT;
	xPreviousBaseValid : BOOL;
	xConfigValid : BOOL;
	xContradiction : BOOL;
	xPairValid : BOOL;
	xWork : BOOL;
	xExchange : BOOL;
	xIdle : BOOL;
	xBase : BOOL;
	xRecovery : BOOL;
	xPneumaticBase : BOOL;
	xPneumaticRecovery : BOOL;
	xManualPneumaticState : BOOL;
	xAutomaticState : BOOL;
	xAxisMotionState : BOOL;
	xManualState : BOOL;
	xAutoSwapAllowed : BOOL;
	xExchangeStartedManual : BOOL; // Обмен начат в ручном режиме: без проверки роботной зоны/точек
	xCommandPresent : BOOL;
	xAccepted : BOOL;
	xStateEntry : BOOL;
	xSeenMotion : BOOL;
	xSeenDone : BOOL;
	xLiftUpCommand : BOOL;
	xLiftDownCommand : BOOL;
	xSelectCommand : BOOL;
	xManualLockCommand : BOOL;
	xManualStopCommand : BOOL;
	xManualLockOutTarget : BOOL;
	xManualStopOutTarget : BOOL;
	xLockOutTarget : BOOL;
	xStopOutTarget : BOOL;
	xStartupInitialized : BOOL;
	xTrustedAtScanStart : BOOL;
	lrWork : LREAL;
	lrTarget : LREAL;
	lrSpan : LREAL;
	rTravel : REAL;
	tStateLimit : TIME;
	tonState : TON;
	tonCoil : TON;
	tonJogLease : TON;
	dwPreviousError : DWORD;
END_VAR
VAR CONSTANT
	ERR_DRIVE : DWORD := DWORD#16#100;
	ERR_SENSOR_CONTRADICTION : DWORD := DWORD#16#200;
	ERR_CYLINDER_TIMEOUT : DWORD := DWORD#16#400;
	ERR_MOTION_TIMEOUT : DWORD := DWORD#16#800;
	ERR_LOGIC : DWORD := DWORD#16#1000;
	ERR_SEQUENCE_INTERRUPTED : DWORD := DWORD#16#2000;
	WRN_COMMAND_REJECTED : UINT := UINT#30;
	WRN_START_REJECTED_BY_OPERATOR : UINT := UINT#31;
	JOG_POSITIVE : UINT := UINT#1;
	JOG_NEGATIVE : UINT := UINT#2;
END_VAR

// --- BEGIN IMPLEMENTATION ---

// Шаги, разрешения и подтверждение положения не восстанавливаются после старта PLC.
IF NOT xStartupInitialized THEN
	Diag.eState := E_TWO_PALLET_STATE.IDLE;
	ePreviousState := E_TWO_PALLET_STATE.IDLE;
	Status.xConfirmed := FALSE;
	Status.xEnabled := FALSE;
	xStartupInitialized := TRUE;
END_IF;

Status.xCompleted := FALSE;
Status.Input := Input;
xTrustedAtScanStart := Status.xConfirmed;

// Все выходные команды импульсные или формируются заново на каждом скане.
Output.xPowerOn := FALSE;
Output.xPowerOff := FALSE;
Output.xDriveReset := FALSE;
Output.xHome := FALSE;
Output.xMove := FALSE;
Output.xStop := FALSE;
Output.xJogPositive := FALSE;
Output.xJogNegative := FALSE;
Output.xTeachOperator := FALSE;
Output.xTeachWork := FALSE;
xLiftUpCommand := FALSE;
xLiftDownCommand := FALSE;
xSelectCommand := FALSE;
xManualLockCommand := FALSE;
xManualStopCommand := FALSE;

// Конфигурация механизма.
xConfigValid := Config.xConfigured
	AND Config.xSignalPatternsConfigured
	AND IsSignalConfigurationValid(uiP1Signals := Config.uiP1Signals, uiP2Signals := Config.uiP2Signals)
	AND (Config.lrTolerance > 0.0)
	AND (Config.lrTolerance <= 20.0)
	AND (ABS(Config.lrWorkP1 - Config.lrExchange) > 2.0 * Config.lrTolerance)
	AND (ABS(Config.lrWorkP2 - Config.lrExchange) > 2.0 * Config.lrTolerance)
	AND ((Config.lrWorkP1 - Config.lrExchange) * (Config.lrWorkP2 - Config.lrExchange) > 0.0)
	AND (Config.lrVelocity > 0.0)
	AND (Config.lrAcceleration > 0.0)
	AND (Config.lrDeceleration > 0.0)
	AND (Config.lrJerk > 0.0)
	AND (Config.tPulse >= T#50MS)
	AND (Config.tCylinder > Config.tPulse)
	AND (Config.tMove > T#0S)
	AND (Config.tHome > T#0S);
Status.xConfigValid := xConfigValid;

// Фактическое состояние пневматики и каретки.
xContradiction := (Input.xLiftUp AND Input.xLiftDown)
	OR (Input.xLockIn AND Input.xLockOut)
	OR (Input.xStopIn AND Input.xStopOut)
	OR (Input.xLimitNegative AND Input.xLimitPositive);
xPairValid := (Input.xLockIn XOR Input.xLockOut)
	AND (Input.xStopIn XOR Input.xStopOut);

uiSignals := UINT#0;
IF Input.xLiftDown THEN uiSignals := uiSignals OR UINT#1; END_IF;
IF Input.xLiftUp THEN uiSignals := uiSignals OR UINT#2; END_IF;
IF Input.xLockIn THEN uiSignals := uiSignals OR UINT#4; END_IF;
IF Input.xLockOut THEN uiSignals := uiSignals OR UINT#8; END_IF;
IF Input.xStopIn THEN uiSignals := uiSignals OR UINT#16; END_IF;
IF Input.xStopOut THEN uiSignals := uiSignals OR UINT#32; END_IF;

uiSelected := UINT#0;
IF xPairValid THEN
	IF (uiSignals AND UINT#60) = (Config.uiP1Signals AND UINT#60) THEN
		uiSelected := UINT#1;
	ELSIF (uiSignals AND UINT#60) = (Config.uiP2Signals AND UINT#60) THEN
		uiSelected := UINT#2;
	END_IF;
END_IF;
xPairValid := xPairValid AND (uiSelected <> UINT#0);

lrWork := Config.lrWorkP1;
uiSelectedSignals := Config.uiP1Signals;
IF uiSelected = UINT#2 THEN
	lrWork := Config.lrWorkP2;
	uiSelectedSignals := Config.uiP2Signals;
END_IF;

xWork := xConfigValid
	AND Input.xHomed
	AND Input.xStandstill
	AND xPairValid
	AND (ABS(Input.lrPosition - lrWork) <= Config.lrTolerance);
xExchange := xConfigValid
	AND Input.xHomed
	AND Input.xStandstill
	AND (ABS(Input.lrPosition - Config.lrExchange) <= Config.lrTolerance);

uiCandidate := UINT#0;
IF xWork
	AND (uiSignals = uiSelectedSignals)
	AND NOT xContradiction
	AND NOT Input.xDriveError
	AND NOT Status.xHomeRequired THEN
	uiCandidate := uiSelected;
END_IF;

xIdle := Diag.eState = E_TWO_PALLET_STATE.IDLE;
xAutomaticState := (Diag.eState = E_TWO_PALLET_STATE.AUTO_LOWER)
	OR (Diag.eState = E_TWO_PALLET_STATE.AUTO_MOVE_TO_EXCHANGE)
	OR (Diag.eState = E_TWO_PALLET_STATE.AUTO_SELECT_PALLET)
	OR (Diag.eState = E_TWO_PALLET_STATE.AUTO_MOVE_TO_WORK)
	OR (Diag.eState = E_TWO_PALLET_STATE.AUTO_RAISE);
xAxisMotionState := (Diag.eState = E_TWO_PALLET_STATE.AUTO_MOVE_TO_EXCHANGE)
	OR (Diag.eState = E_TWO_PALLET_STATE.AUTO_MOVE_TO_WORK)
	OR (Diag.eState = E_TWO_PALLET_STATE.MANUAL_MOVE)
	OR (Diag.eState = E_TWO_PALLET_STATE.MANUAL_HOME)
	OR (Diag.eState = E_TWO_PALLET_STATE.MANUAL_JOG);
xManualState := (Diag.eState = E_TWO_PALLET_STATE.MANUAL_LOWER)
	OR (Diag.eState = E_TWO_PALLET_STATE.MANUAL_RAISE)
	OR (Diag.eState = E_TWO_PALLET_STATE.MANUAL_SELECT_PALLET)
	OR (Diag.eState = E_TWO_PALLET_STATE.MANUAL_MOVE)
	OR (Diag.eState = E_TWO_PALLET_STATE.MANUAL_HOME)
	OR (Diag.eState = E_TWO_PALLET_STATE.MANUAL_JOG)
	OR (Diag.eState = E_TWO_PALLET_STATE.MANUAL_LOCK)
	OR (Diag.eState = E_TWO_PALLET_STATE.MANUAL_STOP);
xManualPneumaticState := (Diag.eState = E_TWO_PALLET_STATE.MANUAL_LOWER)
	OR (Diag.eState = E_TWO_PALLET_STATE.MANUAL_LOCK)
	OR (Diag.eState = E_TWO_PALLET_STATE.MANUAL_STOP);

xBase := xSelected
	AND xConfigValid
	AND Input.xIoMapped
	AND Input.xAxisBound
	AND xSafe
	AND NOT xRobotOperation;
xRecovery := xBase
	AND xManual
	AND xConnection
	AND xIdle
	AND Input.xStandstill;
xPneumaticBase := xSelected
	AND xManual
	AND xSafe
	AND NOT xRobotOperation
	AND Input.xIoMapped
	AND Input.xStandstill;
xPneumaticRecovery := xPneumaticBase AND xIdle;

Status.uiCandidate := uiCandidate;
Status.uiSelected := uiSelected;

// Любое изменение достоверной расстановки аннулирует старое подтверждение.
IF (uiCandidate <> uiPreviousCandidate) OR (xBase <> xPreviousBaseValid) THEN
	Status.udiRevision := Status.udiRevision + UDINT#1;
	IF Status.udiRevision = UDINT#0 THEN
		Status.udiRevision := UDINT#1;
	END_IF;
END_IF;
uiPreviousCandidate := uiCandidate;
xPreviousBaseValid := xBase;

IF xConfigurationChanged THEN
	Status.xConfirmed := FALSE;
	Status.xEnabled := FALSE;
	Status.udiRevision := Status.udiRevision + UDINT#1;
	IF Status.udiRevision = UDINT#0 THEN
		Status.udiRevision := UDINT#1;
	END_IF;
END_IF;

IF NOT xSelected
	OR NOT xSafe
	OR NOT Input.xAxisBound
	OR NOT Input.xIoMapped
	OR NOT xConfigValid
	OR Input.xDriveError
	OR NOT Input.xPowered
	OR (xIdle AND (uiCandidate <> uiConfirmedCandidate)) THEN
	Status.xConfirmed := FALSE;
END_IF;
// Пропадание heartbeat выключает автоматическую обработку, но само по себе
// не перемещает механику и не стирает уже проверенную идентичность палет.
IF NOT xConnection THEN Status.xEnabled := FALSE; END_IF;

// Первая невыполненная предпосылка для HMI.
Diag.uiReason := UINT#0;
IF NOT xSelected THEN
	Diag.uiReason := UINT#1;
ELSIF NOT xConfigValid THEN
	Diag.uiReason := UINT#2;
ELSIF NOT Input.xAxisBound OR NOT Input.xIoMapped THEN
	Diag.uiReason := UINT#3;
ELSIF NOT xSafe THEN
	Diag.uiReason := UINT#4;
ELSIF NOT xConnection THEN
	Diag.uiReason := UINT#17;
ELSIF Input.xDriveError THEN
	Diag.uiReason := UINT#6;
ELSIF Error.dwErrorActive <> DWORD#0 THEN
	Diag.uiReason := UINT#19;
ELSIF NOT Input.xPowered THEN
	Diag.uiReason := UINT#18;
ELSIF xContradiction THEN
	Diag.uiReason := UINT#7;
ELSIF Status.xHomeRequired OR NOT Input.xHomed THEN
	Diag.uiReason := UINT#8;
ELSIF NOT xPairValid THEN
	Diag.uiReason := UINT#9;
ELSIF NOT Input.xStandstill THEN
	Diag.uiReason := UINT#10;
ELSIF NOT xWork THEN
	Diag.uiReason := UINT#11;
ELSIF uiSignals <> uiSelectedSignals THEN
	Diag.uiReason := UINT#12;
ELSIF NOT xIdle THEN
	Diag.uiReason := UINT#22;
ELSIF NOT xRobotMagazineReady THEN
	Diag.uiReason := UINT#16;
ELSIF NOT Status.xConfirmed AND NOT xManual THEN
	Diag.uiReason := UINT#20;
ELSIF NOT Status.xConfirmed THEN
	Diag.uiReason := UINT#13;
END_IF;

// Аварии механизма: биты 8..13 зарезервированы в MAGAZINE_LOGIC_1/2.
IF xSelected AND Input.xDriveError THEN
	Error.dwErrorActive := Error.dwErrorActive OR ERR_DRIVE;
	Status.xHomeRequired := TRUE;
END_IF;

IF xSelected AND xContradiction THEN
	Error.dwErrorActive := Error.dwErrorActive OR ERR_SENSOR_CONTRADICTION;
END_IF;

IF xSelected
	AND NOT xIdle
	AND (((NOT xBase) AND NOT (xManualPneumaticState AND xPneumaticBase))
		OR ((NOT xConnection) AND NOT xManualPneumaticState) OR xStopRequest
		OR (xAutomaticState AND ((xExchangeStartedManual AND (NOT xManual OR NOT xRobotIdle))
			OR (NOT xExchangeStartedManual AND NOT xRobotClear)))) THEN
	Error.dwErrorActive := Error.dwErrorActive OR ERR_SEQUENCE_INTERRUPTED;
	Diag.eState := E_TWO_PALLET_STATE.IDLE;
	Output.xStop := TRUE;
END_IF;

IF xSelected AND (xTrustedAtScanStart OR xAutomaticState) THEN
	IF ((Diag.eState <> E_TWO_PALLET_STATE.AUTO_SELECT_PALLET) AND NOT xPairValid)
		OR (((Diag.eState = E_TWO_PALLET_STATE.AUTO_MOVE_TO_EXCHANGE)
			OR (Diag.eState = E_TWO_PALLET_STATE.AUTO_MOVE_TO_WORK))
			AND (NOT Input.xLiftDown OR Input.xLiftUp))
		OR (xIdle AND (uiCandidate = UINT#0)) THEN
		Error.dwErrorActive := Error.dwErrorActive OR ERR_LOGIC;
	END_IF;
END_IF;

IF xSelected
	AND xTrustedAtScanStart
	AND (NOT xSafe
		OR NOT Input.xAxisBound
		OR NOT Input.xIoMapped
		OR NOT Input.xPowered) THEN
	Error.dwErrorActive := Error.dwErrorActive OR ERR_SEQUENCE_INTERRUPTED;
END_IF;

IF xSelected
	AND ((xContradiction AND NOT xIdle AND NOT xManualPneumaticState)
		OR (Input.xDriveError AND xAxisMotionState)) THEN
	Diag.eState := E_TWO_PALLET_STATE.IDLE;
	Output.xStop := TRUE;
END_IF;

IF xSelected AND NOT Input.xPowered AND (xAutomaticState OR xAxisMotionState) THEN
	Error.dwErrorActive := Error.dwErrorActive OR ERR_SEQUENCE_INTERRUPTED;
	Status.xHomeRequired := TRUE;
	Diag.eState := E_TWO_PALLET_STATE.IDLE;
	Output.xStop := TRUE;
END_IF;

IF Error.dwErrorActive <> DWORD#0 THEN
	Status.xEnabled := FALSE;
	Status.xConfirmed := FALSE;
	IF xAutomaticState THEN
		Diag.eState := E_TWO_PALLET_STATE.IDLE;
		Output.xStop := TRUE;
	END_IF;
END_IF;

// Разрешения считаются только владельцем механизма.
Status.xConfirmAllowed := xRecovery
	AND Input.xPowered
	AND (uiCandidate <> UINT#0)
	AND (Error.dwErrorActive = DWORD#0);
Status.xStartAllowed := Status.xConfirmAllowed
	AND xRobotMagazineReady;
Status.xEnableAllowed := xBase
	AND xConnection
	AND xIdle
	AND Status.xConfirmed
	AND xRobotMagazineReady
	AND (uiCandidate = Status.uiRobotPallet)
	AND Input.xPowered
	AND (Error.dwErrorActive = DWORD#0);
// Операторский обмен выключенного магазина разрешён и в работающем автоцикле.
// В автоматическом режиме требуется окно планировщика и освобождённая зона;
// в ручном режиме остаётся останов робота без проверки его точек/зоны.
Status.xSwapAllowed := xBase
	AND xConnection
	AND xIdle
	AND Input.xStandstill
	AND Input.xPowered
	AND (Error.dwErrorActive = DWORD#0)
	AND Status.xConfirmed
	AND (uiCandidate = Status.uiRobotPallet)
	AND NOT Status.xEnabled
	AND NOT xStopRequest
	AND ((xManual AND xRobotIdle) OR (NOT xManual AND xRobotClear));
xAutoSwapAllowed := Status.xEnableAllowed
	AND xRobotClear
	AND Status.xEnabled
	AND xOtherLoaded;
Status.xPowerAllowed := xRecovery
	AND NOT Input.xDriveError
	AND NOT xContradiction;
Status.xDriveResetAllowed := xSelected
	AND xManual
	AND xConnection
	AND Input.xAxisBound
	AND Input.xStandstill
	AND xIdle;
Status.xLowerAllowed := xPneumaticRecovery;
Status.xRaiseAllowed := xRecovery
	AND NOT xContradiction
	AND NOT Status.xHomeRequired;
Status.xSelectAllowed := xRecovery
	AND NOT xContradiction
	AND Input.xLiftDown
	AND NOT Input.xLiftUp
	AND xExchange;
// Наладочные команды замка и фиксатора независимы от подъёма и координаты.
// Это позволяет вернуть герконы в согласованное состояние после остановки.
Status.xLockAllowed := xPneumaticRecovery;
Status.xStopAllowed := xPneumaticRecovery;
Status.xHomeAllowed := xRecovery
	AND Input.xPowered
	AND NOT Input.xDriveError
	AND Input.xLiftDown
	AND NOT Input.xLiftUp
	AND xPairValid
	AND NOT xContradiction;
Status.xMoveAllowed := Status.xHomeAllowed
	AND Input.xHomed
	AND NOT Status.xHomeRequired;
Status.xJogAllowed := Status.xHomeAllowed;
Status.xTeachOperatorAllowed := Status.xMoveAllowed
	AND Input.xLiftDown
	AND NOT Input.xLiftUp;
Status.xTeachWorkAllowed := Status.xTeachOperatorAllowed
	AND ((uiSelected = UINT#1) OR (uiSelected = UINT#2));
Status.xResetAllowed := xRecovery
	AND (Error.dwErrorActive <> DWORD#0)
	AND NOT xContradiction
	AND NOT Input.xDriveError
	AND NOT Status.xHomeRequired
	AND xPairValid
	AND (Input.xLiftDown XOR Input.xLiftUp);
Status.xConfigAllowed := xSelected
	AND xManual
	AND xIdle
	AND NOT Status.xEnabled
	AND (Input.xStandstill OR NOT Input.xAxisBound)
	AND NOT Input.xPowered
	AND NOT xRobotOperation;

// Командный интерфейс FB не зависит от транспортных номеров HMI 1..19.
xCommandPresent := Command.xEnable
	OR Command.xConfirm
	OR Command.xStart
	OR Command.xRejectStart
	OR Command.xDisable
	OR Command.xSwap
	OR Command.xPowerOn
	OR Command.xPowerOff
	OR Command.xDriveReset
	OR Command.xHome
	OR Command.xLower
	OR Command.xRaise
	OR Command.xSelectPallet
	OR Command.xLockIn
	OR Command.xLockOut
	OR Command.xStopIn
	OR Command.xStopOut
	OR Command.xMoveToExchange
	OR Command.xMoveToWork
	OR Command.xStop
	OR Command.xReset
	OR Command.xJogPositive
	OR Command.xJogNegative
	OR Command.xJogRelease
	OR Command.xTeachOperator
	OR Command.xTeachWork;
xAccepted := NOT xCommandPresent;

IF Command.xStart THEN
	IF Status.xStartAllowed
		AND (Command.udiRevision = Status.udiRevision)
		AND (Command.uiPallet = uiCandidate) THEN
		Status.uiRobotPallet := uiCandidate;
		uiConfirmedCandidate := uiCandidate;
		Status.xConfirmed := TRUE;
		Status.xEnabled := TRUE;
		Status.rP1 := 0.0;
		Status.rP2 := 0.0;
		IF uiCandidate = UINT#1 THEN
			Status.rP1 := 1.0;
		ELSE
			Status.rP2 := 1.0;
		END_IF;
		xAccepted := TRUE;
	END_IF;
ELSIF Command.xRejectStart THEN
	Diag.stWarning.uiCode := WRN_START_REJECTED_BY_OPERATOR;
	Diag.stWarning.udiSequence := Diag.stWarning.udiSequence + UDINT#1;
	IF Diag.stWarning.udiSequence = UDINT#0 THEN
		Diag.stWarning.udiSequence := UDINT#1;
	END_IF;
	xAccepted := TRUE;
ELSIF Command.xEnable THEN
	IF Status.xEnableAllowed THEN
		Status.xEnabled := TRUE;
		xAccepted := TRUE;
	END_IF;
ELSIF Command.xConfirm THEN
	IF Status.xConfirmAllowed
		AND (Command.udiRevision = Status.udiRevision)
		AND (Command.uiPallet = uiCandidate) THEN
		Status.uiRobotPallet := uiCandidate;
		uiConfirmedCandidate := uiCandidate;
		Status.xConfirmed := TRUE;
		Status.rP1 := 0.0;
		Status.rP2 := 0.0;
		IF uiCandidate = UINT#1 THEN
			Status.rP1 := 1.0;
		ELSE
			Status.rP2 := 1.0;
		END_IF;
		xAccepted := TRUE;
	END_IF;
ELSIF Command.xDisable THEN
	Status.xEnabled := FALSE;
	xAccepted := TRUE;
ELSIF Command.xSwap THEN
	IF Status.xSwapAllowed THEN
		xExchangeStartedManual := xManual;
		Diag.eState := E_TWO_PALLET_STATE.AUTO_LOWER;
		xAccepted := TRUE;
	END_IF;
ELSIF Command.xPowerOn THEN
	IF Status.xPowerAllowed THEN
		Output.xPowerOn := TRUE;
		xAccepted := TRUE;
	END_IF;
ELSIF Command.xPowerOff THEN
	IF Status.xDriveResetAllowed THEN
		Output.xPowerOff := TRUE;
		Status.xConfirmed := FALSE;
		Status.xEnabled := FALSE;
		xAccepted := TRUE;
	END_IF;
ELSIF Command.xDriveReset THEN
	IF Status.xDriveResetAllowed AND Input.xDriveError THEN
		Output.xDriveReset := TRUE;
		Status.xConfirmed := FALSE;
		Status.xEnabled := FALSE;
		Status.xHomeRequired := TRUE;
		xAccepted := TRUE;
	END_IF;
ELSIF Command.xHome THEN
	IF Status.xHomeAllowed THEN
		Diag.eState := E_TWO_PALLET_STATE.MANUAL_HOME;
		xAccepted := TRUE;
	END_IF;
ELSIF Command.xLower THEN
	IF Status.xLowerAllowed THEN
		Diag.eState := E_TWO_PALLET_STATE.MANUAL_LOWER;
		xAccepted := TRUE;
	END_IF;
ELSIF Command.xRaise THEN
	IF Status.xRaiseAllowed THEN
		Diag.eState := E_TWO_PALLET_STATE.MANUAL_RAISE;
		xAccepted := TRUE;
	END_IF;
ELSIF Command.xSelectPallet THEN
	IF Status.xSelectAllowed
		AND ((Command.uiPallet = UINT#1) OR (Command.uiPallet = UINT#2)) THEN
		uiTo := Command.uiPallet;
		Diag.eState := E_TWO_PALLET_STATE.MANUAL_SELECT_PALLET;
		xAccepted := TRUE;
	END_IF;
ELSIF Command.xLockIn OR Command.xLockOut THEN
	IF Status.xLockAllowed THEN
		xManualLockOutTarget := Command.xLockOut;
		Diag.eState := E_TWO_PALLET_STATE.MANUAL_LOCK;
		xAccepted := TRUE;
	END_IF;
ELSIF Command.xStopIn OR Command.xStopOut THEN
	IF Status.xStopAllowed THEN
		xManualStopOutTarget := Command.xStopOut;
		Diag.eState := E_TWO_PALLET_STATE.MANUAL_STOP;
		xAccepted := TRUE;
	END_IF;
ELSIF Command.xMoveToExchange OR Command.xMoveToWork THEN
	IF Status.xMoveAllowed THEN
		lrTarget := Config.lrExchange;
		IF Command.xMoveToWork THEN
			lrTarget := lrWork;
		END_IF;
		Diag.eState := E_TWO_PALLET_STATE.MANUAL_MOVE;
		xAccepted := TRUE;
	END_IF;
ELSIF Command.xStop THEN
	Status.xEnabled := FALSE;
	// Stop неподвижного механизма не является ручным вмешательством.
	IF (Diag.eState <> E_TWO_PALLET_STATE.IDLE) OR (Input.xPowered AND NOT Input.xStandstill) THEN
		Output.xStop := TRUE;
		Status.xConfirmed := FALSE;
		Error.dwErrorActive := Error.dwErrorActive OR ERR_SEQUENCE_INTERRUPTED;
	END_IF;
	Diag.eState := E_TWO_PALLET_STATE.IDLE;
	uiJogDirection := UINT#0;
	xAccepted := TRUE;
ELSIF Command.xReset THEN
	IF Status.xResetAllowed THEN
		Error.dwErrorLast := Error.dwErrorActive;
		Error.dwErrorActive := DWORD#0;
		Status.xConfirmed := FALSE;
		Status.xEnabled := FALSE;
		xAccepted := TRUE;
	END_IF;
ELSIF Command.xJogPositive OR Command.xJogNegative THEN
	IF Status.xJogAllowed
		OR ((Diag.eState = E_TWO_PALLET_STATE.MANUAL_JOG)
			AND xBase
			AND xManual
			AND xConnection) THEN
		Diag.eState := E_TWO_PALLET_STATE.MANUAL_JOG;
		IF Command.xJogPositive THEN
			uiJogDirection := JOG_POSITIVE;
		ELSE
			uiJogDirection := JOG_NEGATIVE;
		END_IF;
		xAccepted := TRUE;
	END_IF;
ELSIF Command.xJogRelease THEN
	uiJogDirection := UINT#0;
	IF Diag.eState = E_TWO_PALLET_STATE.MANUAL_JOG THEN
		Diag.eState := E_TWO_PALLET_STATE.IDLE;
		Output.xStop := TRUE;
	END_IF;
	xAccepted := TRUE;
ELSIF Command.xTeachOperator THEN
	IF Status.xTeachOperatorAllowed THEN
		Output.xTeachOperator := TRUE;
		xAccepted := TRUE;
	END_IF;
ELSIF Command.xTeachWork THEN
	IF Status.xTeachWorkAllowed THEN
		Output.xTeachWork := TRUE;
		xAccepted := TRUE;
	END_IF;
END_IF;

IF xCommandPresent AND NOT xAccepted THEN
	Diag.stWarning.uiCode := WRN_COMMAND_REJECTED;
	Diag.stWarning.udiSequence := Diag.stWarning.udiSequence + UDINT#1;
	IF Diag.stWarning.udiSequence = UDINT#0 THEN
		Diag.stWarning.udiSequence := UDINT#1;
	END_IF;
END_IF;

IF xExternalCommandRejected THEN
	Diag.stWarning.uiCode := WRN_COMMAND_REJECTED;
	Diag.stWarning.udiSequence := Diag.stWarning.udiSequence + UDINT#1;
	IF Diag.stWarning.udiSequence = UDINT#0 THEN
		Diag.stWarning.udiSequence := UDINT#1;
	END_IF;
END_IF;

Status.xCommandAccepted := xAccepted;

IF xAutoSwap
	AND xAutoSwapAllowed
	AND NOT Output.xStop
	AND NOT xCommandPresent THEN
	xExchangeStartedManual := FALSE;
	Diag.eState := E_TWO_PALLET_STATE.AUTO_LOWER;
END_IF;

// Стоп ячейки имеет приоритет над командой, принятой в том же скане.
// В IDLE при остановленной оси сохраняем подтверждение и не запускаем MC_Stop.
IF xStopRequest THEN
	IF (Diag.eState <> E_TWO_PALLET_STATE.IDLE) OR (Input.xPowered AND NOT Input.xStandstill) THEN
		Error.dwErrorActive := Error.dwErrorActive OR ERR_SEQUENCE_INTERRUPTED;
		Output.xStop := TRUE;
		Status.xConfirmed := FALSE;
	END_IF;
	Diag.eState := E_TWO_PALLET_STATE.IDLE;
	Status.xEnabled := FALSE;
END_IF;

// Команда могла сменить состояние в этом же скане — обновляем классификацию
// до обработки входа в шаг и запуска таймеров.
xAutomaticState := (Diag.eState = E_TWO_PALLET_STATE.AUTO_LOWER)
	OR (Diag.eState = E_TWO_PALLET_STATE.AUTO_MOVE_TO_EXCHANGE)
	OR (Diag.eState = E_TWO_PALLET_STATE.AUTO_SELECT_PALLET)
	OR (Diag.eState = E_TWO_PALLET_STATE.AUTO_MOVE_TO_WORK)
	OR (Diag.eState = E_TWO_PALLET_STATE.AUTO_RAISE);
xManualState := (Diag.eState = E_TWO_PALLET_STATE.MANUAL_LOWER)
	OR (Diag.eState = E_TWO_PALLET_STATE.MANUAL_RAISE)
	OR (Diag.eState = E_TWO_PALLET_STATE.MANUAL_SELECT_PALLET)
	OR (Diag.eState = E_TWO_PALLET_STATE.MANUAL_MOVE)
	OR (Diag.eState = E_TWO_PALLET_STATE.MANUAL_HOME)
	OR (Diag.eState = E_TWO_PALLET_STATE.MANUAL_JOG)
	OR (Diag.eState = E_TWO_PALLET_STATE.MANUAL_LOCK)
	OR (Diag.eState = E_TWO_PALLET_STATE.MANUAL_STOP);
xManualPneumaticState := (Diag.eState = E_TWO_PALLET_STATE.MANUAL_LOWER)
	OR (Diag.eState = E_TWO_PALLET_STATE.MANUAL_LOCK)
	OR (Diag.eState = E_TWO_PALLET_STATE.MANUAL_STOP);

IF (Diag.eState = E_TWO_PALLET_STATE.AUTO_LOWER)
	AND (ePreviousState <> E_TWO_PALLET_STATE.AUTO_LOWER) THEN
	uiFrom := Status.uiRobotPallet;
	uiTo := UINT#3 - uiFrom;
END_IF;

xStateEntry := Diag.eState <> ePreviousState;
IF xManualState AND xStateEntry THEN
	Status.xConfirmed := FALSE;
	Status.xEnabled := FALSE;
	Status.udiRevision := Status.udiRevision + UDINT#1;
	IF Status.udiRevision = UDINT#0 THEN
		Status.udiRevision := UDINT#1;
	END_IF;
END_IF;

IF xStateEntry THEN
	xSeenMotion := FALSE;
	xSeenDone := FALSE;
	IF (Diag.eState = E_TWO_PALLET_STATE.MANUAL_MOVE)
		OR (Diag.eState = E_TWO_PALLET_STATE.MANUAL_HOME)
		OR (Diag.eState = E_TWO_PALLET_STATE.MANUAL_JOG) THEN
		uiManualSelected := uiSelected;
	END_IF;
ELSIF Input.xMotionDone THEN
	xSeenDone := TRUE;
END_IF;

IF NOT Input.xStandstill THEN
	xSeenMotion := TRUE;
END_IF;

tStateLimit := Config.tCylinder;
IF (Diag.eState = E_TWO_PALLET_STATE.AUTO_MOVE_TO_EXCHANGE)
	OR (Diag.eState = E_TWO_PALLET_STATE.AUTO_MOVE_TO_WORK)
	OR (Diag.eState = E_TWO_PALLET_STATE.MANUAL_MOVE) THEN
	tStateLimit := Config.tMove;
END_IF;
IF Diag.eState = E_TWO_PALLET_STATE.MANUAL_HOME THEN
	tStateLimit := Config.tHome;
END_IF;

tonState(
	IN := NOT xIdle
		AND (Diag.eState <> E_TWO_PALLET_STATE.MANUAL_JOG)
		AND NOT xStateEntry,
	PT := tStateLimit);
tonCoil(
	IN := NOT xIdle AND NOT xStateEntry,
	PT := Config.tPulse);
tonJogLease(
	IN := (Diag.eState = E_TWO_PALLET_STATE.MANUAL_JOG)
		AND NOT (Command.xJogPositive OR Command.xJogNegative),
	PT := T#350MS);
ePreviousState := Diag.eState;

// Автомат обмена и ручного восстановления.
uiTargetSignals := Config.uiP1Signals;
IF uiTo = UINT#2 THEN uiTargetSignals := Config.uiP2Signals; END_IF;
CASE Diag.eState OF
	E_TWO_PALLET_STATE.AUTO_LOWER,
	E_TWO_PALLET_STATE.MANUAL_LOWER:
		xLiftDownCommand := TRUE;
		IF Input.xLiftDown AND NOT Input.xLiftUp THEN
			IF Diag.eState = E_TWO_PALLET_STATE.AUTO_LOWER THEN
				Diag.eState := E_TWO_PALLET_STATE.AUTO_MOVE_TO_EXCHANGE;
				lrTarget := Config.lrExchange;
			ELSE
				Diag.eState := E_TWO_PALLET_STATE.IDLE;
			END_IF;
		END_IF;

	E_TWO_PALLET_STATE.AUTO_MOVE_TO_EXCHANGE,
	E_TWO_PALLET_STATE.AUTO_MOVE_TO_WORK,
	E_TWO_PALLET_STATE.MANUAL_MOVE:
		IF Diag.eState = E_TWO_PALLET_STATE.AUTO_MOVE_TO_WORK THEN
			lrTarget := Config.lrWorkP1;
			IF uiTo = UINT#2 THEN
				lrTarget := Config.lrWorkP2;
			END_IF;
		END_IF;

		IF NOT Input.xLiftDown
			OR Input.xLiftUp
			OR NOT xPairValid
			OR Status.xHomeRequired
			OR ((Diag.eState = E_TWO_PALLET_STATE.AUTO_MOVE_TO_EXCHANGE) AND (uiSelected <> uiFrom))
			OR ((Diag.eState = E_TWO_PALLET_STATE.AUTO_MOVE_TO_WORK) AND (uiSelected <> uiTo))
			OR ((Diag.eState = E_TWO_PALLET_STATE.MANUAL_MOVE) AND (uiSelected <> uiManualSelected))
			OR (Input.xLimitPositive AND (lrTarget > Input.lrPosition + Config.lrTolerance))
			OR (Input.xLimitNegative AND (lrTarget < Input.lrPosition - Config.lrTolerance)) THEN
			Error.dwErrorActive := Error.dwErrorActive OR ERR_LOGIC;
			Diag.eState := E_TWO_PALLET_STATE.IDLE;
			Output.xStop := TRUE;
		ELSE
			Output.lrTarget := lrTarget;
			Output.xMove := xStateEntry;
			IF Input.xStandstill
				AND (ABS(Input.lrPosition - lrTarget) <= Config.lrTolerance)
				AND ((xSeenMotion OR xSeenDone) OR xStateEntry) THEN
				Output.xMove := FALSE;
				IF Diag.eState = E_TWO_PALLET_STATE.AUTO_MOVE_TO_EXCHANGE THEN
					Diag.eState := E_TWO_PALLET_STATE.AUTO_SELECT_PALLET;
				ELSIF Diag.eState = E_TWO_PALLET_STATE.AUTO_MOVE_TO_WORK THEN
					Diag.eState := E_TWO_PALLET_STATE.AUTO_RAISE;
				ELSE
					Diag.eState := E_TWO_PALLET_STATE.IDLE;
				END_IF;
			END_IF;
		END_IF;

	E_TWO_PALLET_STATE.AUTO_SELECT_PALLET,
	E_TWO_PALLET_STATE.MANUAL_SELECT_PALLET:
		IF NOT xExchange OR NOT Input.xLiftDown OR Input.xLiftUp THEN
			Error.dwErrorActive := Error.dwErrorActive OR ERR_LOGIC;
			Diag.eState := E_TWO_PALLET_STATE.IDLE;
			Output.xStop := TRUE;
		ELSE
			xSelectCommand := TRUE;
		END_IF;
		IF (uiSelected = uiTo) AND xPairValid AND NOT Output.xStop THEN
			IF Diag.eState = E_TWO_PALLET_STATE.AUTO_SELECT_PALLET THEN
				Diag.eState := E_TWO_PALLET_STATE.AUTO_MOVE_TO_WORK;
			ELSE
				Diag.eState := E_TWO_PALLET_STATE.IDLE;
			END_IF;
		END_IF;

	E_TWO_PALLET_STATE.MANUAL_LOCK:
		IF xManualLockOutTarget THEN
			xManualLockCommand := NOT Input.xLockOut OR Input.xLockIn;
			IF Input.xLockOut AND NOT Input.xLockIn THEN Diag.eState := E_TWO_PALLET_STATE.IDLE; END_IF;
		ELSE
			xManualLockCommand := NOT Input.xLockIn OR Input.xLockOut;
			IF Input.xLockIn AND NOT Input.xLockOut THEN Diag.eState := E_TWO_PALLET_STATE.IDLE; END_IF;
		END_IF;

	E_TWO_PALLET_STATE.MANUAL_STOP:
		IF xManualStopOutTarget THEN
			xManualStopCommand := NOT Input.xStopOut OR Input.xStopIn;
			IF Input.xStopOut AND NOT Input.xStopIn THEN Diag.eState := E_TWO_PALLET_STATE.IDLE; END_IF;
		ELSE
			xManualStopCommand := NOT Input.xStopIn OR Input.xStopOut;
			IF Input.xStopIn AND NOT Input.xStopOut THEN Diag.eState := E_TWO_PALLET_STATE.IDLE; END_IF;
		END_IF;

	E_TWO_PALLET_STATE.AUTO_RAISE:
		// Завершение обмена устанавливает подъём по выбранной конфигурации
		// только после фактического останова в рабочей позиции.
		IF NOT xWork
			OR Status.xHomeRequired
			OR (uiSelected <> uiTo) THEN
			Error.dwErrorActive := Error.dwErrorActive OR ERR_LOGIC;
			Diag.eState := E_TWO_PALLET_STATE.IDLE;
			Output.xStop := TRUE;
		ELSE
			xLiftUpCommand := (uiTargetSignals AND UINT#2) <> UINT#0;
			xLiftDownCommand := NOT xLiftUpCommand;
			IF uiSignals = uiTargetSignals THEN
				Status.uiRobotPallet := uiTo;
				uiConfirmedCandidate := uiTo;
				Status.xConfirmed := TRUE;
				Status.xCompleted := TRUE;
				Diag.eState := E_TWO_PALLET_STATE.IDLE;
			END_IF;
		END_IF;

	E_TWO_PALLET_STATE.MANUAL_RAISE:
		// Наладочный подъём не требует HOME-координаты или рабочей позиции.
		IF NOT Input.xStandstill OR NOT xManual OR xContradiction OR Status.xHomeRequired THEN
			Error.dwErrorActive := Error.dwErrorActive OR ERR_LOGIC;
			Diag.eState := E_TWO_PALLET_STATE.IDLE;
			Output.xStop := TRUE;
		ELSE
			xLiftUpCommand := TRUE;
			IF Input.xLiftUp AND NOT Input.xLiftDown THEN
				Diag.eState := E_TWO_PALLET_STATE.IDLE;
			END_IF;
		END_IF;

	E_TWO_PALLET_STATE.MANUAL_HOME:
		Output.xHome := xStateEntry;
		IF xSeenDone
			AND Input.xHomed
			AND Input.xStandstill
			AND NOT xStateEntry THEN
			Status.xHomeRequired := FALSE;
			Diag.eState := E_TWO_PALLET_STATE.IDLE;
		END_IF;

	E_TWO_PALLET_STATE.MANUAL_JOG:
		IF tonJogLease.Q OR NOT xConnection OR (uiJogDirection = UINT#0) THEN
			Diag.eState := E_TWO_PALLET_STATE.IDLE;
			Output.xStop := TRUE;
		ELSE
			Output.xJogPositive := (uiJogDirection = JOG_POSITIVE) AND NOT Input.xLimitPositive;
			Output.xJogNegative := (uiJogDirection = JOG_NEGATIVE) AND NOT Input.xLimitNegative;
		END_IF;

	E_TWO_PALLET_STATE.IDLE:
		uiJogDirection := UINT#0;

ELSE
	Error.dwErrorActive := Error.dwErrorActive OR ERR_LOGIC;
	Diag.eState := E_TWO_PALLET_STATE.IDLE;
	Output.xStop := TRUE;
END_CASE;
IF Diag.eState = E_TWO_PALLET_STATE.IDLE THEN xExchangeStartedManual := FALSE; END_IF;

// Низ П2 и выбранное зацепление контролируются всё время Home/JOG.
IF ((Diag.eState = E_TWO_PALLET_STATE.MANUAL_HOME)
	OR (Diag.eState = E_TWO_PALLET_STATE.MANUAL_JOG))
	AND (NOT Input.xLiftDown
		OR Input.xLiftUp
		OR NOT xPairValid
		OR (uiSelected <> uiManualSelected)
		OR xContradiction
		OR Input.xDriveError
		OR NOT Input.xPowered) THEN
	Error.dwErrorActive := Error.dwErrorActive OR ERR_LOGIC;
	Diag.eState := E_TWO_PALLET_STATE.IDLE;
	Output.xStop := TRUE;
END_IF;

IF tonState.Q THEN
	IF (ePreviousState = E_TWO_PALLET_STATE.AUTO_MOVE_TO_EXCHANGE)
		OR (ePreviousState = E_TWO_PALLET_STATE.AUTO_MOVE_TO_WORK)
		OR (ePreviousState = E_TWO_PALLET_STATE.MANUAL_MOVE)
		OR (ePreviousState = E_TWO_PALLET_STATE.MANUAL_HOME) THEN
		Error.dwErrorActive := Error.dwErrorActive OR ERR_MOTION_TIMEOUT;
		Status.xHomeRequired := TRUE;
	ELSE
		Error.dwErrorActive := Error.dwErrorActive OR ERR_CYLINDER_TIMEOUT;
	END_IF;
	Diag.eState := E_TWO_PALLET_STATE.IDLE;
	Output.xStop := TRUE;
END_IF;

IF (((NOT xBase) AND NOT (xManualPneumaticState AND xPneumaticBase))
	OR ((NOT xConnection) AND NOT xManualPneumaticState))
	AND (ePreviousState <> E_TWO_PALLET_STATE.IDLE)
	OR Output.xStop THEN
	Output.xMove := FALSE;
	Output.xHome := FALSE;
	Output.xJogPositive := FALSE;
	Output.xJogNegative := FALSE;
	xLiftUpCommand := FALSE;
	xLiftDownCommand := FALSE;
	xSelectCommand := FALSE;
	xManualLockCommand := FALSE;
	xManualStopCommand := FALSE;
END_IF;

// Автоматический обмен переключает пару совместно; ручное восстановление — каждый цилиндр отдельно.
xLockOutTarget := (uiTargetSignals AND UINT#8) <> UINT#0;
xStopOutTarget := (uiTargetSignals AND UINT#32) <> UINT#0;
Output.xLiftUp := xBase AND xLiftUpCommand AND NOT tonCoil.Q;
Output.xLiftDown := (xBase OR xPneumaticBase) AND xLiftDownCommand AND NOT tonCoil.Q;
Output.xLockOut := (xBase AND xSelectCommand AND xLockOutTarget
	OR xPneumaticBase AND xManualLockCommand AND xManualLockOutTarget) AND NOT tonCoil.Q;
Output.xLockIn := (xBase AND xSelectCommand AND NOT xLockOutTarget
	OR xPneumaticBase AND xManualLockCommand AND NOT xManualLockOutTarget) AND NOT tonCoil.Q;
Output.xStopOut := (xBase AND xSelectCommand AND xStopOutTarget
	OR xPneumaticBase AND xManualStopCommand AND xManualStopOutTarget) AND NOT tonCoil.Q;
Output.xStopIn := (xBase AND xSelectCommand AND NOT xStopOutTarget
	OR xPneumaticBase AND xManualStopCommand AND NOT xManualStopOutTarget) AND NOT tonCoil.Q;

// Поза для 3D — оценка по координате каретки и подтверждённому зацеплению.
IF xPairValid AND Input.xHomed THEN
	lrSpan := lrWork - Config.lrExchange;
	IF ABS(lrSpan) > Config.lrTolerance THEN
		rTravel := LREAL_TO_REAL(
			LIMIT(0.0, (Input.lrPosition - Config.lrExchange) / lrSpan, 1.0));
		IF uiSelected = UINT#1 THEN
			Status.rP1 := rTravel;
		ELSE
			Status.rP2 := rTravel;
		END_IF;
	END_IF;
END_IF;

IF Input.xLiftUp AND NOT Input.xLiftDown THEN
	Status.rLift := 1.0;
ELSIF Input.xLiftDown AND NOT Input.xLiftUp THEN
	Status.rLift := 0.0;
END_IF;

// Диагностика и совместимый публичный Status формируются в одном месте.
IF (Error.dwErrorActive <> dwPreviousError)
	AND (Error.dwErrorActive <> DWORD#0) THEN
	Diag.eFaultState := ePreviousState;
END_IF;
dwPreviousError := Error.dwErrorActive;

IF Error.dwErrorActive <> DWORD#0 THEN
	Error.dwErrorLast := Error.dwErrorActive;
	Status.xConfirmed := FALSE;
	Status.xEnabled := FALSE;
END_IF;
Error.dwAlarmActive := Error.dwErrorActive;
Error.stErrorActive := UpdateErrorView(dwError := Error.dwErrorActive);
Error.stErrorLast := UpdateErrorView(dwError := Error.dwErrorLast);

Status.uiStep := TO_UINT(Diag.eState);
Status.uiFaultStep := TO_UINT(Diag.eFaultState);
Status.uiReason := Diag.uiReason;
Status.dwError := Error.dwErrorActive;
Status.stWarning := Diag.stWarning;
Status.xBusy := Diag.eState <> E_TWO_PALLET_STATE.IDLE;
Status.xError := Error.dwErrorActive <> DWORD#0;

// Команда или автомат могли занять механизм после первоначального расчёта
// разрешений. Не публикуем устаревшее разрешение ещё на один скан.
IF Status.xBusy THEN
	Status.xConfirmAllowed := FALSE;
	Status.xStartAllowed := FALSE;
	Status.xEnableAllowed := FALSE;
	Status.xSwapAllowed := FALSE;
	Status.xPowerAllowed := FALSE;
	Status.xDriveResetAllowed := FALSE;
	Status.xHomeAllowed := FALSE;
	Status.xLowerAllowed := FALSE;
	Status.xRaiseAllowed := FALSE;
	Status.xSelectAllowed := FALSE;
	Status.xLockAllowed := FALSE;
	Status.xStopAllowed := FALSE;
	Status.xMoveAllowed := FALSE;
	Status.xJogAllowed := FALSE;
	Status.xTeachOperatorAllowed := FALSE;
	Status.xTeachWorkAllowed := FALSE;
	Status.xResetAllowed := FALSE;
	Status.xConfigAllowed := FALSE;
END_IF;

// Инвентарь операторской палеты редактируется всегда, независимо от режима,
// движения, подтверждения, питания и ошибок механизма. Роботная палета — только
// при выключенном магазине после освобождения текущей/выданной операции с ним.
// Считаем после команд и обмена, чтобы роль палеты была актуальна в этом скане.
Status.xEdit1Allowed := xSelected
	AND ((Status.uiRobotPallet <> UINT#1) OR (NOT Status.xEnabled AND xActivePalletEditAllowed));
Status.xEdit2Allowed := xSelected
	AND ((Status.uiRobotPallet <> UINT#2) OR (NOT Status.xEnabled AND xActivePalletEditAllowed));
Status.xEditAllowed := Status.xEdit1Allowed OR Status.xEdit2Allowed;

Status.xReady := xSelected
	AND Status.xEnabled
	AND Status.xConfirmed
	AND NOT Status.xBusy
	AND NOT Status.xError
	AND xWork
	AND (uiCandidate = Status.uiRobotPallet)
	AND Input.xPowered
	AND xRobotGeometryReady
	AND xRobotMagazineReady
	AND xSafe
	AND xConnection;

IF NOT xSelected THEN
	Status.xEnabled := FALSE;
	Status.xConfirmed := FALSE;
END_IF;

(* ---- FB_TWO_PALLET_SIMULATION.st ---- *)
FUNCTION_BLOCK FB_TWO_PALLET_SIMULATION
VAR_INPUT
	xEnable : BOOL; // Только тестовая среда SIMULATION
	uiP1Signals : UINT;
	Command : ST_TWO_PALLET_OUTPUT;
END_VAR
VAR_OUTPUT
	xLiftDown : BOOL;
	xLiftUp : BOOL;
	xLockIn : BOOL;
	xLockOut : BOOL;
	xStopIn : BOOL;
	xStopOut : BOOL;
END_VAR
VAR
	xInitialized : BOOL;
	xLiftTargetUp : BOOL;
	xLockTargetOut : BOOL;
	xStopTargetOut : BOOL;
	tonLift : TON;
	tonLock : TON;
	tonStop : TON;
END_VAR

// --- BEGIN IMPLEMENTATION ---

IF NOT xEnable THEN
	xInitialized := FALSE;
	xLiftDown := FALSE;
	xLiftUp := FALSE;
	xLockIn := FALSE;
	xLockOut := FALSE;
	xStopIn := FALSE;
	xStopOut := FALSE;
	tonLift(IN := FALSE, PT := T#300MS);
	tonLock(IN := FALSE, PT := T#300MS);
	tonStop(IN := FALSE, PT := T#300MS);
ELSE
	IF NOT xInitialized THEN
		// Виртуальная начальная поза: П2 внизу, замок держит П1,
		// фиксатор держит противоположную палету.
		xLiftTargetUp := FALSE;
		xLockTargetOut := (uiP1Signals AND UINT#8) <> UINT#0;
		xStopTargetOut := (uiP1Signals AND UINT#32) <> UINT#0;
		xLiftDown := TRUE;
		xLiftUp := FALSE;
		xLockOut := xLockTargetOut;
		xLockIn := NOT xLockTargetOut;
		xStopOut := xStopTargetOut;
		xStopIn := NOT xStopTargetOut;
		xInitialized := TRUE;
	END_IF;

	// Бистабильный 5/2 сохраняет положение после снятия обеих катушек.
	IF Command.xLiftUp AND NOT Command.xLiftDown THEN
		xLiftTargetUp := TRUE;
	ELSIF Command.xLiftDown AND NOT Command.xLiftUp THEN
		xLiftTargetUp := FALSE;
	END_IF;
	IF Command.xLockOut AND NOT Command.xLockIn THEN
		xLockTargetOut := TRUE;
	ELSIF Command.xLockIn AND NOT Command.xLockOut THEN
		xLockTargetOut := FALSE;
	END_IF;
	IF Command.xStopOut AND NOT Command.xStopIn THEN
		xStopTargetOut := TRUE;
	ELSIF Command.xStopIn AND NOT Command.xStopOut THEN
		xStopTargetOut := FALSE;
	END_IF;

	tonLift(IN := xLiftTargetUp <> xLiftUp, PT := T#300MS);
	tonLock(IN := xLockTargetOut <> xLockOut, PT := T#300MS);
	tonStop(IN := xStopTargetOut <> xStopOut, PT := T#300MS);
	IF tonLift.Q THEN
		xLiftUp := xLiftTargetUp;
		xLiftDown := NOT xLiftTargetUp;
	END_IF;
	IF tonLock.Q THEN
		xLockOut := xLockTargetOut;
		xLockIn := NOT xLockTargetOut;
	END_IF;
	IF tonStop.Q THEN
		xStopOut := xStopTargetOut;
		xStopIn := NOT xStopTargetOut;
	END_IF;
END_IF;

(* ---- FB_ALARM_MANAGER.AddEvent.st ---- *)
METHOD PRIVATE AddEvent
VAR_INPUT
	eSource   : E_ALARM_SOURCE; // Источник события
	eSeverity : E_ALARM_SEVERITY; // Уровень события
	uiCode    : UINT; // Код события внутри источника
END_VAR

// --- BEGIN IMPLEMENTATION ---

udiSequence := udiSequence + 1;
IF udiSequence = UDINT#0 THEN
	udiSequence := UDINT#1;
END_IF;

Events[uiWriteIndex].udiSequence := udiSequence;
Events[uiWriteIndex].eSeverity := eSeverity;
Events[uiWriteIndex].eSource := eSource;
Events[uiWriteIndex].uiCode := uiCode;
Events[uiWriteIndex].xActive := TRUE;

IF uiWriteIndex >= 100 THEN
	uiWriteIndex := 1;
ELSE
	uiWriteIndex := uiWriteIndex + 1;
END_IF;

(* ---- FB_ALARM_MANAGER.DeactivateEvent.st ---- *)
METHOD PRIVATE DeactivateEvent
VAR_INPUT
	eSource : E_ALARM_SOURCE; // Источник аварии
	uiCode  : UINT; // Номер очищенного бита
END_VAR
VAR
	uiIndex : UINT; // Индекс поиска в журнале
END_VAR

// --- BEGIN IMPLEMENTATION ---

FOR uiIndex := 1 TO 100 DO
	IF Events[uiIndex].xActive
	AND (Events[uiIndex].eSeverity = E_ALARM_SEVERITY.ALARM)
	AND (Events[uiIndex].eSource = eSource)
	AND (Events[uiIndex].uiCode = uiCode) THEN
		Events[uiIndex].xActive := FALSE;
	END_IF;
END_FOR;

(* ---- FB_ALARM_MANAGER.GetAlarmEffect.st ---- *)
METHOD PRIVATE GetAlarmEffect : E_ALARM_EFFECT
VAR_INPUT
	eSource : E_ALARM_SOURCE; // Первичный владелец ошибки
	uiCode : UINT; // Номер бита ошибки владельца
	xRobotStopRequired : BOOL; // Защёлкнутый контекст оборудования требует остановить робота
	xGlobalError : BOOL; // Активна Safety-ошибка ячейки
END_VAR

// --- BEGIN IMPLEMENTATION ---

// Safety имеет абсолютный приоритет над любой частной причиной.
IF xGlobalError THEN
	GetAlarmEffect := E_ALARM_EFFECT.GLOBAL_STOP;

ELSE
CASE eSource OF
	E_ALARM_SOURCE.CELL_SAFETY:
		GetAlarmEffect := E_ALARM_EFFECT.GLOBAL_STOP;

	E_ALARM_SOURCE.CELL:
		CASE uiCode OF
			1: GetAlarmEffect := E_ALARM_EFFECT.ROBOT_STOP; // ERR_ROBOT
			4: GetAlarmEffect := E_ALARM_EFFECT.GLOBAL_STOP; // ERR_GLOBAL_STOP
		ELSE GetAlarmEffect := E_ALARM_EFFECT.EQUIPMENT_STOP;
		END_CASE;

	E_ALARM_SOURCE.MACHINE_1,
	E_ALARM_SOURCE.MACHINE_2,
	E_ALARM_SOURCE.MACHINE_3:
		CASE uiCode OF
			9: GetAlarmEffect := E_ALARM_EFFECT.GLOBAL_STOP; // ERR_SAFETY_STOP
			2, 3, 13, 15, 16, 17, 23: GetAlarmEffect := E_ALARM_EFFECT.ROBOT_STOP;
		ELSE
			IF xRobotStopRequired THEN
				GetAlarmEffect := E_ALARM_EFFECT.ROBOT_STOP;
			ELSE
				GetAlarmEffect := E_ALARM_EFFECT.EQUIPMENT_STOP;
			END_IF;
		END_CASE;

	E_ALARM_SOURCE.MAGAZINE_LOGIC_1,
	E_ALARM_SOURCE.MAGAZINE_LOGIC_2:
		CASE uiCode OF
			5: GetAlarmEffect := E_ALARM_EFFECT.ROBOT_STOP; // ERR_ROBOT
			6: GetAlarmEffect := E_ALARM_EFFECT.GLOBAL_STOP; // ERR_GLOBAL_STOP
		ELSE
			IF xRobotStopRequired THEN
				GetAlarmEffect := E_ALARM_EFFECT.ROBOT_STOP;
			ELSE
				GetAlarmEffect := E_ALARM_EFFECT.EQUIPMENT_STOP;
			END_IF;
		END_CASE;

	E_ALARM_SOURCE.RESERVED_LEGACY_MAGAZINE_AXIS_1,
	E_ALARM_SOURCE.RESERVED_LEGACY_MAGAZINE_AXIS_2:
		IF xRobotStopRequired THEN
			GetAlarmEffect := E_ALARM_EFFECT.ROBOT_STOP;
		ELSE
			GetAlarmEffect := E_ALARM_EFFECT.EQUIPMENT_STOP;
		END_IF;

	E_ALARM_SOURCE.ROBOT,
	E_ALARM_SOURCE.AXIS_X,
	E_ALARM_SOURCE.AXIS_Y,
	E_ALARM_SOURCE.AXIS_Z,
	E_ALARM_SOURCE.AXIS_GROUP,
	E_ALARM_SOURCE.MOTION_MANAGER,
	E_ALARM_SOURCE.POINT_MANAGER,
	E_ALARM_SOURCE.GRIPPER:
		GetAlarmEffect := E_ALARM_EFFECT.ROBOT_STOP;

ELSE
	GetAlarmEffect := E_ALARM_EFFECT.EQUIPMENT_STOP;
END_CASE;
END_IF;

(* ---- FB_ALARM_MANAGER.UpdateSource.st ---- *)
METHOD PRIVATE UpdateSource
VAR_INPUT
	eSource   : E_ALARM_SOURCE; // Источник проверяемой маски ошибок
	dwCurrent : DWORD; // Текущая маска ошибок
END_VAR
VAR_IN_OUT
	dwPrevious : DWORD; // Маска ошибок прошлого цикла
END_VAR
VAR
	dwChanged : DWORD; // Изменившиеся биты
	dwBit     : DWORD; // Маска проверяемого бита
	uiBit     : UINT; // Номер проверяемого бита
END_VAR

// --- BEGIN IMPLEMENTATION ---

dwChanged := dwCurrent XOR dwPrevious;

IF dwChanged <> DWORD#0 THEN
	FOR uiBit := 0 TO 31 DO
		dwBit := SHL(DWORD#1, uiBit);
		IF (dwChanged AND dwBit) <> DWORD#0 THEN
			IF (dwCurrent AND dwBit) <> DWORD#0 THEN
				AddEvent(eSource := eSource, eSeverity := E_ALARM_SEVERITY.ALARM, uiCode := uiBit);
			ELSE
				DeactivateEvent(eSource := eSource, uiCode := uiBit);
			END_IF;
		END_IF;
	END_FOR;
	dwPrevious := dwCurrent;
END_IF;

(* ---- FB_AXIS.UpdateErrorView.st ---- *)
METHOD UpdateErrorView : ST_AXIS_ERROR
VAR_INPUT
	dwAxisError   : DWORD; // Маска ошибок SoftMotion и привода
	dwLogicalError: DWORD; // Маска логических ошибок оси
END_VAR
VAR
	stError : ST_AXIS_ERROR; // Представление ошибок отдельными флагами
END_VAR

// --- BEGIN IMPLEMENTATION ---

stError.MC_POWER_ERROR := (dwAxisError AND AXE_MC_POWER_ERROR) <> DWORD#0;
stError.MC_RESET_ERROR := (dwAxisError AND AXE_MC_RESET_ERROR) <> DWORD#0;
stError.MC_STOP_ERROR := (dwAxisError AND AXE_MC_STOP_ERROR) <> DWORD#0;
stError.MC_JOG_ERROR := (dwAxisError AND AXE_MC_JOG_ERROR) <> DWORD#0;
stError.MC_HOME_ERROR := (dwAxisError AND AXE_MC_HOME_ERROR) <> DWORD#0;
stError.MC_MOVE_ABS_ERROR := (dwAxisError AND AXE_MC_MOVE_ABS_ERROR) <> DWORD#0;
stError.MC_MOVE_REL_ERROR := (dwAxisError AND AXE_MC_MOVE_REL_ERROR) <> DWORD#0;
stError.READ_POSITION_ERROR := (dwAxisError AND AXE_READ_POS_ERROR) <> DWORD#0;
stError.READ_STATUS_ERROR := (dwAxisError AND AXE_READ_STATUS_ERROR) <> DWORD#0;
stError.AXIS_ERRORSTOP := (dwAxisError AND AXE_ERRORSTOP) <> DWORD#0;
stError.FB_ERROR_OCCURRED := (dwAxisError AND AXE_FB_ERROR_OCCURRED) <> DWORD#0;
stError.COMMAND_ABORTED := (dwAxisError AND AXE_COMMAND_ABORTED) <> DWORD#0;
stError.UNKNOWN_AXIS_ERROR := (dwAxisError AND AXE_UNKNOWN_ACTUAL_ERROR) <> DWORD#0;
stError.DRIVE_AXIS_ERROR := (dwAxisError AND AXE_DRIVE_AXIS_ERROR) <> DWORD#0;
stError.POWER_FEEDBACK_LOST := (dwAxisError AND AXE_POWER_FEEDBACK_LOST) <> DWORD#0;

stError.POWER_PERMIT_LOST := (dwLogicalError AND LOG_POWER_PERMIT_LOST) <> DWORD#0;
stError.GLOBAL_DURING_POWER := (dwLogicalError AND LOG_GLOBAL_DURING_POWER) <> DWORD#0;
stError.GLOBAL_DURING_READY := (dwLogicalError AND LOG_GLOBAL_DURING_READY) <> DWORD#0;
stError.GLOBAL_DURING_MOTION := (dwLogicalError AND LOG_GLOBAL_DURING_MOTION) <> DWORD#0;
stError.JOG_CONFLICT := (dwLogicalError AND LOG_JOG_CONFLICT) <> DWORD#0;
stError.MOVE_ABS_NOT_HOMED := (dwLogicalError AND LOG_MOVE_ABS_NOT_HOMED) <> DWORD#0;
stError.MOVE_REL_NOT_HOMED := (dwLogicalError AND LOG_MOVE_REL_NOT_HOMED) <> DWORD#0;
stError.STEP_TIMEOUT := (dwLogicalError AND LOG_STEP_TIMEOUT) <> DWORD#0;
stError.UNKNOWN_STEP := (dwLogicalError AND LOG_UNKNOWN_STEP) <> DWORD#0;

UpdateErrorView := stError;

(* ---- FB_AXIS_GROUP.UpdateErrorView.st ---- *)
METHOD UpdateErrorView : ST_AXIS_GROUP_ERROR
VAR_INPUT
	dwMotionError : DWORD; // Маска ошибок блоков SoftMotion
	dwLogicalError: DWORD; // Маска логических ошибок группы
END_VAR
VAR
	stError : ST_AXIS_GROUP_ERROR; // Представление ошибок отдельными флагами
END_VAR

// --- BEGIN IMPLEMENTATION ---

stError.ENABLE_ERROR := (dwMotionError AND MOTION_ERR_ENABLE) <> DWORD#0;
stError.POWER_ERROR := (dwMotionError AND MOTION_ERR_POWER) <> DWORD#0;
stError.DISABLE_ERROR := (dwMotionError AND MOTION_ERR_DISABLE) <> DWORD#0;
stError.RESET_ERROR := (dwMotionError AND MOTION_ERR_RESET) <> DWORD#0;
stError.MOVE_DIRECT_ERROR := (dwMotionError AND MOTION_ERR_MOVE_DIRECT) <> DWORD#0;
stError.MOVE_LINEAR_ERROR := (dwMotionError AND MOTION_ERR_MOVE_LINEAR) <> DWORD#0;
stError.HALT_ERROR := (dwMotionError AND MOTION_ERR_HALT) <> DWORD#0;
stError.STOP_ERROR := (dwMotionError AND MOTION_ERR_STOP) <> DWORD#0;
stError.READ_POSITION_ERROR := (dwMotionError AND MOTION_ERR_READ_POSITION) <> DWORD#0;
stError.READ_STATUS_ERROR := (dwMotionError AND MOTION_ERR_READ_STATUS) <> DWORD#0;
stError.READ_GROUP_ERROR := (dwMotionError AND MOTION_ERR_READ_GROUP_ERROR) <> DWORD#0;
stError.GROUP_ERROR_STOP := (dwMotionError AND MOTION_ERR_GROUP_ERROR_STOP) <> DWORD#0;

stError.STEP_TIMEOUT := (dwLogicalError AND LOG_STEP_TIMEOUT) <> DWORD#0;
stError.INVALID_STATE := (dwLogicalError AND LOG_INVALID_STATE) <> DWORD#0;
stError.POWER_PERMIT_READY := (dwLogicalError AND LOG_POWER_PERMIT_READY) <> DWORD#0;
stError.POWER_PERMIT_LOST := (dwLogicalError AND LOG_POWER_PERMIT_LOST_DIRECT) <> DWORD#0;

UpdateErrorView := stError;

(* ---- FB_CELL_MANAGER.UpdateErrorView.st ---- *)
METHOD UpdateErrorView : ST_CELL_ERROR
VAR_INPUT
	dwError : DWORD; // Битовая маска для расшифровки
END_VAR
VAR
	stError : ST_CELL_ERROR; // Представление ошибок отдельными флагами
END_VAR

// --- BEGIN IMPLEMENTATION ---

stError.BOTH_GRIPPERS_OCCUPIED := (dwError AND ERR_BOTH_GRIPPERS) <> DWORD#0;
stError.ROBOT_ERROR := (dwError AND ERR_ROBOT) <> DWORD#0;
stError.MAGAZINE_ERROR := (dwError AND ERR_MAGAZINE) <> DWORD#0;
stError.MACHINE_ERROR := (dwError AND ERR_MACHINE) <> DWORD#0;
stError.GLOBAL_STOP := (dwError AND ERR_GLOBAL_STOP) <> DWORD#0;

UpdateErrorView := stError;

(* ---- FB_CELL_SAFETY.RaiseWarning.st ---- *)
METHOD PRIVATE RaiseWarning
VAR_INPUT
	uiCode : UINT;
END_VAR

// --- BEGIN IMPLEMENTATION ---

Diag.stWarning.uiCode := uiCode;
Diag.stWarning.udiSequence := Diag.stWarning.udiSequence + UDINT#1;
IF Diag.stWarning.udiSequence = UDINT#0 THEN
	Diag.stWarning.udiSequence := UDINT#1;
END_IF;

(* ---- FB_GRIPPER_SIMULATION.UpdateErrorView.st ---- *)
METHOD UpdateErrorView : ST_GRIPPER_ERROR
VAR_INPUT
	dwError : DWORD; // Битовая маска для расшифровки
END_VAR
VAR
	stError : ST_GRIPPER_ERROR; // Представление ошибок отдельными флагами
END_VAR

// --- BEGIN IMPLEMENTATION ---

stError.GRIPPER_1_ERROR := (dwError AND ERR_GRIPPER_1) <> DWORD#0;
stError.GRIPPER_2_ERROR := (dwError AND ERR_GRIPPER_2) <> DWORD#0;
stError.ROTATION_ERROR := (dwError AND ERR_GRIP_ROTATE) <> DWORD#0;
stError.ACTION_ERROR := (dwError AND ERR_GRIP_ACTION) <> DWORD#0;
stError.GLOBAL_ERROR := (dwError AND ERR_GRIP_GLOBAL) <> DWORD#0;

UpdateErrorView := stError;

(* ---- FB_MACHINE.UpdateErrorView.st ---- *)
METHOD UpdateErrorView : ST_MACHINE_ERROR
VAR_INPUT
	dwError : DWORD; // Битовая маска для расшифровки
END_VAR
VAR
	stError : ST_MACHINE_ERROR; // Представление ошибок отдельными флагами
END_VAR

// --- BEGIN IMPLEMENTATION ---

stError.WRONG_OPERATION := (dwError AND ERR_WRONG_OPERATION) <> DWORD#0;
stError.WRONG_COMMAND := (dwError AND ERR_WRONG_COMMAND) <> DWORD#0;
stError.ROBOT_MOTION := (dwError AND ERR_ROBOT_MOTION) <> DWORD#0;
stError.ROBOT_ACTION := (dwError AND ERR_ROBOT_ACTION) <> DWORD#0;
stError.DOOR_OPEN := (dwError AND ERR_DOOR_OPEN) <> DWORD#0;
stError.DOOR_CLOSE := (dwError AND ERR_DOOR_CLOSE) <> DWORD#0;
stError.CHUCK_OPEN := (dwError AND ERR_CHUCK_OPEN) <> DWORD#0;
stError.CHUCK_CLOSE := (dwError AND ERR_CHUCK_CLOSE) <> DWORD#0;
stError.CYCLE_START := (dwError AND ERR_CYCLE_START) <> DWORD#0;
stError.SAFETY_STOP := (dwError AND ERR_SAFETY_STOP) <> DWORD#0;
stError.UNKNOWN_DETAIL := (dwError AND ERR_UNKNOWN_DETAIL) <> DWORD#0;
stError.MACHINE_ALARM := (dwError AND ERR_MACHINE_ALARM) <> DWORD#0;
stError.INDEX_ERROR := (dwError AND ERR_INDEX) <> DWORD#0;
stError.DOOR_ROBOT := (dwError AND ERR_DOOR_ROBOT) <> DWORD#0;
stError.MACHINE_IDLE := (dwError AND ERR_MACHINE_IDLE) <> DWORD#0;
stError.TIMEOUT_ROBOT_MOVE := (dwError AND ERR_TIMEOUT_ROBOT_MOVE) <> DWORD#0;
stError.TIMEOUT_ROBOT_ACTION := (dwError AND ERR_TIMEOUT_ROBOT_ACTION) <> DWORD#0;
stError.TIMEOUT_ROBOT_RELEASE := (dwError AND ERR_TIMEOUT_ROBOT_RELEASE) <> DWORD#0;
stError.TIMEOUT_DOOR_OPEN := (dwError AND ERR_TIMEOUT_DOOR_OPEN) <> DWORD#0;
stError.TIMEOUT_DOOR_CLOSE := (dwError AND ERR_TIMEOUT_DOOR_CLOSE) <> DWORD#0;
stError.TIMEOUT_HATCH_UNLOCK := (dwError AND ERR_TIMEOUT_HATCH_UNLOCK) <> DWORD#0;
stError.TIMEOUT_CHUCK_OPEN := (dwError AND ERR_TIMEOUT_CHUCK_OPEN) <> DWORD#0;
stError.TIMEOUT_CHUCK_CLOSE := (dwError AND ERR_TIMEOUT_CHUCK_CLOSE) <> DWORD#0;
stError.TIMEOUT_CYCLE_START := (dwError AND ERR_TIMEOUT_CYCLE_START) <> DWORD#0;
stError.SAFETY_DOOR_OPEN := (dwError AND ERR_SAFETY_DOOR_OPEN) <> DWORD#0;
stError.HATCH_UNLOCK_PROCESSING := (dwError AND ERR_HATCH_UNLOCK_PROCESSING) <> DWORD#0;

UpdateErrorView := stError;

(* ---- FB_MAGAZINE.FindBlank.st ---- *)
METHOD FindBlank : SINT
VAR_INPUT
	iSlotCount : SINT; // Число слотов, участвующих в поиске
END_VAR
VAR_IN_OUT
	stDetail : ARRAY [1..GVL_CELL_SETTINGS.NumberDetail] OF ST_DETAIL; // Содержимое слотов магазина
END_VAR
VAR
	i : SINT; // Индекс проверяемого слота
END_VAR

// --- BEGIN IMPLEMENTATION ---

FindBlank := 0;

FOR i:= 1 TO iSlotCount DO
	IF stDetail[i].xInPosition = TRUE AND stDetail[i].eDetailType =  E_DETAIL_TYPE.BLANK THEN
		FindBlank := i;
		EXIT;
	END_IF
END_FOR

(* ---- FB_MAGAZINE.FindFreeSlot.st ---- *)
METHOD FindFreeSlot : SINT
VAR_INPUT
	iSlotCount : SINT; // Число слотов, участвующих в поиске
END_VAR
VAR_IN_OUT
	stDetail : ARRAY [1..GVL_CELL_SETTINGS.NumberDetail] OF ST_DETAIL; // Содержимое слотов магазина
END_VAR
VAR
	i : SINT; // Индекс проверяемого слота
END_VAR

// --- BEGIN IMPLEMENTATION ---

FindFreeSlot := 0;

FOR i:= 1 TO iSlotCount DO
	IF stDetail[i].xInPosition = FALSE THEN
		FindFreeSlot := i;
		EXIT;
	END_IF
END_FOR
